(* CODESYS project CtaAppSensor_2.0.0.0.library
   Description: Sensor Library der CTA
   Version: 2.0.0.0
   Title: CtaAppSensor
   Author: SIS
   DocFormat: reStructuredText
   Placeholder: CtaAppSensor
   LanguageModelAttribute: qualified-access-only
   CompiledLibraryCompatibilityVersion: CODESYS V3.5 SP16 Patch 3
   Company: CTA
   DefaultNamespace: CtaAppSensor

Project tree, tasks and I/O mapping:
  libraries: Standard, 3.5.18.0 (System); CtaAppBmk, 2.0.0.0 (CTA); CtaAppReport, 2.0.0.0 (CTA); CtaSysConfig, 2.0.0.0 (CTA); CtaAppFilter, 1.0.0.0 (CTA); VisuSymbols, 4.5.0.0 (System); VisuDialogs, * (System); CtaSysSensorReCalculation, 1.0.0.0 (CTA); CtaVisSymbols, 2.0.0.0 (CTA); CtaAppInfluxLog, 1.0.0.1 (CTA); CtaSysIO, 2.0.0.0 (CTA); CtaVisHelp, 2.0.0.0 (CTA); CtaAppModbusSpezifikation, 1.0.0.1 (CTA); CtaVisApps, 1.0.0.0 (CTA); CtaSysFU, 2.0.0.0 (CTA)
  40 Visualizations/
    ICON/
      SENSOR_FLAT/
        SENSOR_FLAT_TXT_RIGHT/
          ABOVE/
            visualisation VIS_SENSOR_FLAT_RigthAboveCheckIsEnabled
            visualisation VIS_SENSOR_FLAT_RIGHT_ABOVE
            visualisation VIS_SENSOR_FLAT_RigthAboveCheckQuerry
          BELOW/
            visualisation VIS_SENSOR_FLAT_RIGHT_BELOW
            visualisation VIS_SENSOR_FLAT_RigthBelowCheckIsEnabled
            visualisation VIS_SENSOR_FLAT_RigthBelowCheckQuerry
          MIDDLE/
            visualisation VIS_SENSOR_FLAT_RIGHT_MIDDLE
            visualisation VIS_SENSOR_FLAT_RigthMiddleCheckIsEnabled
            visualisation VIS_SENSOR_FLAT_RigthMiddleCheckQuerry
        SENSOR_FLAT_TXT_LEFT/
          BELOW/
            visualisation VIS_SENSOR_FLAT_LEFT_BELOW
            visualisation VIS_SENSOR_FLAT_LeftBelowCheckIsEnabled
            visualisation VIS_SENSOR_FLAT_LeftBelowCheckQuerry
          ABOVE/
            visualisation VIS_SENSOR_FLAT_LeftAboveCheckQuerry
            visualisation VIS_SENSOR_FLAT_LEFT_ABOVE
            visualisation VIS_SENSOR_FLAT_LeftAboveCheckIsEnabled
          MIDDLE/
            visualisation VIS_SENSOR_FLAT_LeftMiddleCheckIsEnabled
            visualisation VIS_SENSOR_FLAT_LeftMiddleCheckQuerry
            visualisation VIS_SENSOR_FLAT_LEFT_MIDDLE
      SENSOR_BASE/
        ICON/
          Round/
            visualisation SensorRound
          Flat/
            visualisation SensorFlat
          Value/
            visualisation ValueDwnUp
            visualisation ValueUpDwn
      SENSOR_ROUND/
        SENSOR_ROUND_TXT_RIGHT/
          ABOVE/
            visualisation VIS_SENSOR_ROUND_RIGHT_ABOVE
            visualisation VIS_SENSOR_ROUND_RightAboveCheckIsEnabled
            visualisation VIS_SENSOR_ROUND_RightAboveCheckQuerry
          BELOW/
            visualisation VIS_SENSOR_ROUND_RIGHT_BELOW
            visualisation VIS_SENSOR_ROUND_RightBelowCheckQuerry
            visualisation VIS_SENSOR_ROUND_RightBelowCheckIsEnabled
        SENSOR_ROUNF_TXT_LEFT/
          ABOVE/
            visualisation VIS_SENSOR_ROUND_LEFT_ABOVE
            visualisation VIS_SENSOR_ROUND_LeftAboveCheckIsEnabled
            visualisation VIS_SENSOR_ROUND_LeftAboveCheckQuerry
          BELOW/
            visualisation VIS_SENSOR_ROUND_LEFT_BELOW
            visualisation VIS_SENSOR_ROUND_LeftBelowCheckIsEnabled
            visualisation VIS_SENSOR_ROUND_LeftBelowCheckQuerry
    POPUP/
      visualisation POPUP_SENSOR
      PARAMETER/
        visualisation VIS_SENSOR_PARAMETER
        visualisation VIS_SENSOR_PARAMETER_LISTE
        SENSOR_ParameterBase/
          visualisation VIS_SENSOR_PARAMETER_BASE0
          visualisation VIS_SENSOR_PARAMETER_BASE
        SENSOR_ReportManagement/
          visualisation Sensor_LowAlarm_Param
          visualisation Sensor_HighAlarm_Param
          visualisation Sensor_HighWarning_Param
          visualisation VIS_SENSOR_PARAMETER_REPORTMNG
          visualisation VIS_SENSOR_PARAMETER_REPORTMNG_1
          visualisation Sensor_LowWarning_Param
        SENSOR_InfluxDb/
          visualisation VIS_SENSOR_PARAMETER_TRENDLOG
          visualisation VIS_SENSOR_PARAMETER_TRENDLOG0
        SENSOR_Filter/
          visualisation VIS_SENSOR_PARAMETER_FILTER
          visualisation VIS_SENSOR_PARAMETER_FILTER_1
        IO_Parameter/
          visualisation VIS_SENSOR_IO_PARAMETER
      visualisation VIS_SENSOR_LISTE
      MANUAL/
        visualisation VIS_SENSOR_MANUAL
      OVERVIEW/
        visualisation VIS_SENSOR_OVERVIEW
        visualisation VIS_SENSOR_OVERVIEW0
      REPORTS/
        visualisation VIS_SENSOR_REPORTS
      BUS/
        visualisation Sensor_BUS_CS
        visualisation Sensor_BUS
        visualisation Sensor_BUS_SW0_Detail
        visualisation Sensor_BUS_SW1_Detail
        visualisation Sensor_BUS_SW2_Detail
        visualisation Sensor_BUS_SW3_Detail
      PLACEHOLDER/
        visualisation VIS_SENSOR_PLACEHOLDER
        visualisation VIS_SENSOR_PLACEHOLDER0
        visualisation VIS_SENSOR_PLACEHOLDER_1
        visualisation VIS_SENSOR_PLACEHOLDER0_1
  30 Program Organization Units/
    fb's/
      Sensor/
        function block fbSensor [ST]: proModulType, actReport, proITF_REPORTMANAGER, actErrorCondition, proLockDown, proAvailable, proAcknowlege, proAtIconNr, actTrendLog, proEn, proEnSymbol, metSetReal, metSetBool, proIsEnabled, proIsError, proStateSymbol, proCountedError, proCountedInfo, proCountedWarning, actState, proInvertierung, proxErrorConditionValue, proConfigError, actConfig, P_scAnalogAlarm_fbxEnableOverflowAl, P_scAnalogAlarm_fbxEnableUnderflowAl, P_scBase_fbxEnable, P_scVisu_fbusiDezimalPos, P_scAlCondition_fbxEnable, P_scAlCondition_fbtDelayTillCondition, P_scHighAlarm_fbiRetryTillLock, P_scHighAlarm_fbiTypeOfAcknolage, P_scHighAlarm_fbrHysterese, P_scHighAlarm_fbrValue, P_scHighAlarm_fbtDelayTillAlarm, P_scHighAlram_fbxDoesAlarm, P_scHighWarning_fbrValue, P_scHighWarning_fbtDelayTillWarning, P_scHighWarning_fbxDoesWarning, P_scInfluxDb_fbxEnable, P_scLoAlarm_fbiRetryTillLock, P_scLoAlarm_fbiTypeOfAcknolage, P_scLoAlarm_fbrHysterese, P_scLoAlarm_fbrValue, P_scLoAlarm_fbtDelayTillAlarm, P_scLoAlarm_fbxDoesAlarm, P_scLoWarning_fbrValue, P_scLoWarning_fbtDelayTillWarning, P_scLoWarning_fbxDoesWarning, P_scManual_fbrManualOnY, P_scManual_fbuiManualControl, P_scManual_fbuiManualState, P_scManual_fbxAllowManualOn, P_scAlarmReset_fbtDealyTillReset, P_scFilter_fbrValue, P_scFilter_fbxEnabled, proSensorITF, proRawValue, proSoftwareValue, proIsWarning, proIsHandOnOrOff, proIsReady, proHandOff, proHandOn, proHandOnY, proAuto, proManualTrue, proManualFalse, proValueInputType, metSetITF, actDigital, actAnalog, proPhysicalValue, actReCalculate, ITF_RC, actMbState, proModbusTest, proModbusStateWord, proModbusControllWord, prorValue
    fc's/
      function fcGetBigerStringValue [ST]
      AlarmControll/
        function fcHighControl [ST]
        function fcLowControl [ST]
      Visu/
        function fcCheckQuerryAndIconReturn [ST]
  00000000-0000-0000-0000-000000000000|D:\CoDeSys\LibrariesV3\trunk\Intern\CAA\CAA Template\3.4.0.0 draft\Placeholder.xml
  00000000-0000-0000-0000-000000000000|D:\CoDeSys\LibrariesV3\trunk\Intern\CAA\CAA Template\3.2.0.3 draft\Prefix.pdf
  00000000-0000-0000-0000-000000000000|D:\CoDeSys\LibrariesV3\trunk\Intern\CAA\CAA Template\3.5.2.0 draft\Placeholder.xml
  20 Structs/
    data type scParameter
    LowWarning/
      data type scLoWarning
    BASE/
      data type scBase
    Alarme/
      data type scAnalogAlarm
      Zusatzbedingungen/
        data type scAlCondition
      AlarmReset/
        data type scAlarmReset
    HighWarning/
      data type scHighWarning
    InfluxDb/
      data type scInfluxDb
    Filter/
      data type scFilter
    HighAlarm/
      data type scHighAlarm
    LowAlarm/
      data type scLoAlarm
    Manual/
      data type scManual
    data type enInputType
    Visu/
      data type scVisu
  50 Images/
  10 Documenation/
    global variables VersionHistory
    global variables readMe
  21 Interface/
    interface ITF_SENSOR: proConfigError, P_scBase_fbxEnable, P_scVisu_fbusiDezimalPos, P_scManual_fbxAllowManualOn, P_scManual_fbuiManualState, P_scManual_fbuiManualControl, P_scManual_fbrManualOnY, P_scFilter_fbxEnabled, P_scFilter_fbrValue, P_scLoWarning_fbxDoesWarning, P_scLoWarning_fbrValue, P_scLoWarning_fbtDelayTillWarning, P_scLoAlarm_fbxDoesAlarm, P_scLoAlarm_fbrValue, P_scLoAlarm_fbrHysterese, P_scLoAlarm_fbtDelayTillAlarm, P_scLoAlarm_fbiRetryTillLock, P_scLoAlarm_fbiTypeOfAcknolage, P_scHighWarning_fbxDoesWarning, P_scHighWarning_fbrValue, P_scHighWarning_fbtDelayTillWarning, P_scHighAlram_fbxDoesAlarm, P_scHighAlarm_fbrValue, P_scHighAlarm_fbrHysterese, P_scHighAlarm_fbtDelayTillAlarm, P_scHighAlarm_fbiRetryTillLock, P_scHighAlarm_fbiTypeOfAcknolage, P_scInfluxDb_fbxEnable, P_scAnalogAlarm_fbxEnableOverflowAl, P_scAnalogAlarm_fbxEnableUnderflowAl, P_scAlCondition_fbxEnable, P_scAlCondition_fbtDelayTillCondition, P_scAlarmReset_fbtDealyTillReset, proSensorITF, proCountedError, proCountedInfo, proITF_REPORTMANAGER, proCountedWarning, proRawValue, proSoftwareValue, proEnSymbol, proStateSymbol, proIsHandOnOrOff, proHandOn, proIsError, proIsWarning, proEn, proIsEnabled, proHandOff, proHandOnY, proIsReady, proAuto, proManualFalse, proManualTrue, proValueInputType, proPhysicalValue, proxErrorConditionValue, proInvertierung, prorValue, proLockDown, proAvailable, proAcknowlege, proAtIconNr, ITF_RC, proModbusStateWord, proModbusTest, proModbusControllWord
  11 Library Parameter/
  12 Konstanten/
    global variables GlobalKonstant
  60 Textlisten/
    text list GlobalTextList
    text list Info
    Types/
      text list WarnungsStatus
      text list ValueInputType
    Reports/
      text list Error
      text list Warnung
  13 Globale Variablen/
  5ce3da45-db07-42e7-a21c-a00fff4ed8f6|C:\Users\sis\Downloads\dip-switch.svg
  5ce3da45-db07-42e7-a21c-a00fff4ed8f6|C:\Users\sis\Downloads\lightning-bolt-circle.svg
  5ce3da45-db07-42e7-a21c-a00fff4ed8f6|C:\Users\sis\Downloads\sine-wave.svg
  5ce3da45-db07-42e7-a21c-a00fff4ed8f6|C:\Users\sis\Downloads\eye.svg
  5ce3da45-db07-42e7-a21c-a00fff4ed8f6|C:\Users\sis\Downloads\lan.svg
*)

// 20 Structs/scParameter
{attribute 'pack_mode' := '1'} 
TYPE scParameter :
    STRUCT
        scBase              :   scBase;
		scManual			:	scManual;
		scFilter			:	scFilter;
		scLoWarning			:	scLoWarning;
		scLoAlarm			:	scLoAlarm;
		scHighWarning		:	scHighWarning;
		scHighAlarm			:	scHighAlarm;
		scInfluxDb			:	scInfluxDb;
		scAnalogAlarm		:	scAnalogAlarm;
		scAlCondition		:	scAlCondition;
		scAlarmReset		:	scAlarmReset;
		scVisu				:	scVisu;
    END_STRUCT
END_TYPE

// 20 Structs/HighWarning/scHighWarning
TYPE scHighWarning :
	STRUCT
		fbxDoesWarning			:	CtaSysConfig.fbBOOL;
		fbrValue				:	CtaSysConfig.fbREAL;
		fbtDelayTillWarning		:	CtaSysConfig.fbTIME;	
	END_STRUCT
END_TYPE

// 20 Structs/HighAlarm/scHighAlarm
TYPE scHighAlarm :
	STRUCT
		fbxDoesAlarm			:	CtaSysConfig.fbBOOL;
		fbrValue				:	CtaSysConfig.fbREAL;
		fbrHysterese			:	CtaSysConfig.fbREAL;
		fbtDeleayTillAlarm		:	CtaSysConfig.fbTIME;
		fbiRetryTillLock		:	CtaSysConfig.fbINT;
		fbiTypeOfAcknolage		:	CtaSysConfig.fbINT;
	END_STRUCT
END_TYPE

// 20 Structs/LowAlarm/scLoAlarm
TYPE scLoAlarm :
	STRUCT
		fbxDoesAlarm			:	CtaSysConfig.fbBOOL;
		fbrValue				:	CtaSysConfig.fbREAL;
		fbrHysterese			:	CtaSysConfig.fbREAL;
		fbtDeleayTillAlarm		:	CtaSysConfig.fbTIME;
		fbiRetryTillLock		:	CtaSysConfig.fbINT;
		fbiTypeOfAcknolage		:	CtaSysConfig.fbINT;
	END_STRUCT
END_TYPE

// 20 Structs/LowWarning/scLoWarning
TYPE scLoWarning :
	STRUCT
		fbxDoesWarning			:	CtaSysConfig.fbBOOL;
		fbrValue				:	CtaSysConfig.fbREAL;
		fbtDelayTillWarning		:	CtaSysConfig.fbTIME;		
	END_STRUCT
END_TYPE

// 20 Structs/Alarme/scAnalogAlarm
TYPE scAnalogAlarm :
	STRUCT
		fbxEnableOverflowAl		:	CtaSysConfig.fbBOOL;
		fbxEnableUnderflowAl	:	CtaSysConfig.fbBOOL;
	END_STRUCT
END_TYPE

// 20 Structs/Filter/scFilter
TYPE scFilter :
	STRUCT
		fbxEnabled	:	CtaSysConfig.fbBOOL;
		fbrValue	:	CtaSysConfig.fbREAL;
	END_STRUCT
END_TYPE

// 20 Structs/BASE/scBase
{attribute 'pack_mode' := '1'} 
TYPE scBase :
    STRUCT
        fbxEnable       :   CtaSysConfig.fbBOOL;
    END_STRUCT
END_TYPE

// 20 Structs/InfluxDb/scInfluxDb
{attribute 'pack_mode' := '1'} 
TYPE scInfluxDb :
    STRUCT
        fbxEnable       :   CtaSysConfig.fbBOOL;
    END_STRUCT
END_TYPE

// 20 Structs/Alarme/Zusatzbedingungen/scAlCondition
TYPE scAlCondition :
	STRUCT
		fbxEnable				:	CtaSysConfig.fbBOOL;
		fbtDelayTillCondition	:	CtaSysConfig.fbTIME;
	END_STRUCT
END_TYPE

// 20 Structs/Alarme/AlarmReset/scAlarmReset
TYPE scAlarmReset :
	STRUCT
		fbtDelayTillReset	:	CtaSysConfig.fbTIME;		
	END_STRUCT
END_TYPE

// 20 Structs/Manual/scManual
TYPE scManual :
	STRUCT
		fbxAlowManualOn		:	CtaSysConfig.fbBOOL;
		fbuiManualState		:	CtaSysConfig.fbUINT;
		fbuiManualControl	:	CtaSysConfig.fbUINT;
		fbrManualOnY		:	CtaSysConfig.fbREAL;
	END_STRUCT
END_TYPE

// 20 Structs/enInputType
{attribute 'qualified_only'}
{attribute 'strict'}
TYPE enInputType :
(
	Default := 0,
	AnalogInput,
	DigitalInput,
	Analog_ITF_Input,
	Digital_ITF_Input	
);
END_TYPE

// 20 Structs/Visu/scVisu
TYPE scVisu :
	STRUCT
		fbusiDezimalPos		:	CtaSysConfig.fbUSINT;
	END_STRUCT
END_TYPE

// 10 Documenation/VersionHistory
(* 

.. image:: ../../Images/CTA_Logo.jpg
   :align: right
   :width: 15% 

**Vorlage**   


============ =========== =========== ============================================
**Date**     **Version** **Author**  **Change**
------------ ----------- ----------- --------------------------------------------
04.03.2021   0.0.0.0     SIS         Vorlage erstellt

============ =========== =========== ============================================


*)
VAR_GLOBAL
    stInfo : STRING:= '0.0.0.0, Vorlage, CTA';
END_VAR

// 10 Documenation/readMe
(*

**ReadMe**
 
|	**Empfehlung**
|
|	Bibliothek CtaAppSensor zur auswertung von Sensoren
|	Instanzieren Sie den CtaAppSensor.fbSensor in ihrem Funktionsbaustein oder POU beispielsweise als fbTFühlX (X = Nr.) 
|	Deklarieren Sie die Struktur Variable welche als Parameter und zur ansteuerung dienen wie im Code beispiel.
|  
| *Beispiel* 

+-----------------------+---------------------------------------------------------------------------------------------------------------------------------------------------------------------------------------------------------------------------------------------------------------------------------------------------------------------------------------------------------------------------------------------------------------------------------------+
| Beschreibung          |  Code                                                                                                                                                                                                                                                                                                                                                                                                                                 |
+=======================+=======================================================================================================================================================================================================================================================================================================================================================================================================================================+
| POU oder SmFb         | .. code-block:: codesys                                                                                                                                                                                                                                                                                                                                                                                                               |
|                       |                                                                                                                                                                                                                                                                                                                                                                                                                                       |
|                       |	// Deklaration als VAR im POU oder dem selbsterstellten Funktionsbaustein                                                                                                                                                                                                                                                                                                                                                        	|
|                       |   VAR   																																																				 																																																				|
|						|	    (*Temperaturfühler 1*)																																																		 																																																	|
|						|		fbTFühl1			: CtaAppSensor.fbSensor;                                                                                                                                                                                                                                                                                                                                                               						|
|			 			|	END_VAR                                                                                                                                                                                                                                                                                                                                                                                                                          	|
+-----------------------+---------------------------------------------------------------------------------------------------------------------------------------------------------------------------------------------------------------------------------------------------------------------------------------------------------------------------------------------------------------------------------------------------------------------------------------+
| Code für Init         | .. code-block:: codesys                                                                                                                                                                                                                                                                                                                                                                                                               |
|                       |   																																																					 																																																				|
|			 			|	// Kopieren des nachfolgenden Codes in eine Action zur Initialisierung der Parameter. Zum Beispiel actConfig.																																																				 																										|
|                       |	{region "Parameter Temperaturfühler 1"}                                                                                                                                                                                                                                                                                                                                                                                             |
|			 			|		(*Basis*)                                                                                                                                                                                                                                                                                                                                                                                                                       |
|						|		fbTFühl1.scParameter.scBase.fbxEnable                			(_WertInit :=  TRUE																		 );		//P1 Ein- Ausschalten des Sensors                                                                                                                                                                                                                               |
|						|		(*Handansteuerung*)                                                                                                                                                                                                                                                                                                                                                                                                             |
|						|		fbTFühl1.scParameter.scManual.fbxAlowManualOn					(_WertInit := FALSE																		 );     //P2 Handansteuerung zulassen / nicht zulassen                                                                                                                                                                                                                  |
|						|		fbTFühl1.scParameter.scManual.fbuiManualState					(_WertInit :=	  0									, _MinInit :=     0, _MaxInit:=     2);     //P3 Ansteuerungsmodus des Sensors (auto, manuell, gesperrt)                                                                                                                                                                                                    |
|						|		fbTFühl1.scParameter.scManual.fbuiManualControl					(_WertInit :=     0									, _MinInit :=     0, _MaxInit:=     1);     //P4 Ansteuerungsignal des Sensors (TRUE,FALSE)                                                                                                                                                                                                                 |
|						|		fbTFühl1.scParameter.scManual.fbrManualOnY						(_WertInit :=   0.0									, _MinInit :=      , _MaxInit:=      );     //P5 Manueller Stellwert für den SEnsor                                                                                                                                                                                                                         |
|						|		(*Filter*)                                                                                                                                                                                                                                                                                                                                                                                                                      |
|						|		fbTFühl1.scParameter.scFilter.fbxEnabled						(_WertInit := FALSE																		 );		//P6 Ein- Ausschalten des Filters                                                                                                                                                                                                                               |
|						|		fbTFühl1.scParameter.scFilter.fbrValue							(_WertInit :=   0.0									, _MinInit :=      , _MaxInit:=      );		//P7 Filterwert                                                                                                                                                                                                                                                 |
|						|		(*LowWarning*)                                                                                                                                                                                                                                                                                                                                                                                                                  |
|						|		fbTFühl1.scParameter.scLoWarning.fbxDoesWarning					(_WertInit := FALSE																		 );		//P8 Ein- Ausschalten der LowWarning                                                                                                                                                                                                                            |
|						|		fbTFühl1.scParameter.scLoWarning.fbrValue						(_WertInit :=   0.0									, _minInit :=      , _maxInit:= 	 );		//P9 Wert bei welcher die LowWarning ausgelöst wird                                                                                                                                                                                                             |
|						|		fbTFühl1.scParameter.scLoWarning.fbtDelayTillWarning			(_WertInit :=  T#0S									, _minInit :=      , _maxInit:=      );		//P10 Verzögerungszeit für die Ausgabe des LowWarining Fehlers                                                                                                                                                                                                  |
|						|		(*LowAlarm*)                                                                                                                                                                                                                                                                                                                                                                                                                    |
|						|		fbTFühl1.scParameter.scLoAlarm.fbxDoesAlarm						(_WertInit := FALSE																		 );		//P11 Ein- Ausschalten des LowAlarm                                                                                                                                                                                                                             |
|						|		fbTFühl1.scParameter.scLoAlarm.fbrValue							(_WertInit :=   0.0									, _minInit :=      , _maxInit:= 	 );		//P12 Wert bei welchem der LowAlarm ausgelöst wird                                                                                                                                                                                                              |
|						|		fbTFühl1.scParameter.scLoAlarm.fbrHysterese						(_WertInit :=   0.0									, _minInit :=      , _maxInit:= 	 );		//P13 Histerese welche zur Rücksetung des Fehlers erreicht werden muss                                                                                                                                                                                          |
|						|		fbTFühl1.scParameter.scLoAlarm.fbtDeleayTillAlarm				(_WertInit :=  T#0S									, _minInit :=      , _maxInit:= 	 );		//P14 Verzögerungszeit für die Ausgabe des LowAlarm Fehlers                                                                                                                                                                                                     |
|						|		fbTFühl1.scParameter.scLoAlarm.fbiTypeOfAcknolage				(_WertInit :=     0 								, _minInit :=     0, _maxInit:=     2);		//P15 Art der Quittierung des Fehlers (auto, quittierned, quittiernd bis n Meldung)                                                                                                                                                                             |
|						|		fbTFühl1.scParameter.scLoAlarm.fbiRetryTillLock					(_WertInit :=     3									, _minInit :=     0, _maxInit:=     5);		//P16 Maximale Anzahl Wiederholungen bis zu Sperrung der Anlage                                                                                                                                                                                                 |
|						|		(*HighWarning*)                                                                                                                                                                                                                                                                                                                                                                                                                 |
|						|		fbTFühl1.scParameter.scHighWarning.fbxDoesWarning				(_WertInit := FALSE																		 );		//P17 Ein- Ausschalten der HighWarning                                                                                                                                                                                                                    		|
|						|		fbTFühl1.scParameter.scHighWarning.fbrValue						(_WertInit :=   0.0									, _minInit :=      , _maxInit:= 	 );		//P18 Wert bei welcher die HighWarning ausgelöst wird                                                                                                                                                                                                     		|
|						|		fbTFühl1.scParameter.scHighWarning.fbtDelayTillWarning			(_WertInit :=  T#0S									, _minInit := 	   , _maxInit:= 	 );		//P19 Verzögerungszeit für die Ausgabe des HighWarining Fehlers                                                                                                                                                                                           		|
|						|		(*HighAlarm*)                                                                                                                                                                                                                                                                                                                                                                                                                   |
|						|		fbTFühl1.scParameter.scHighAlarm.fbxDoesAlarm					(_WertInit := FALSE															 			 );		//P20 Ein- Ausschalten des HighAlarm                                                                                                                                                                                                                            |
|						|		fbTFühl1.scParameter.scHighAlarm.fbrValue						(_WertInit :=   0.0									, _minInit :=      , _maxInit:=      );		//P21 Wert bei welchem der HighAlarm ausgelöst wird                                                                                                                                                                                                             |
|						|		fbTFühl1.scParameter.scHighAlarm.fbrHysterese					(_WertInit :=   0.0									, _minInit :=      , _maxInit:= 	 );		//P22 Histerese welche zur Rücksetung des Fehlers erreicht werden muss                                                                                                                                                                                          |
|						|		fbTFühl1.scParameter.scHighAlarm.fbtDeleayTillAlarm				(_WertInit :=  T#0S									, _minInit :=      , _maxInit:=      );		//P23 Verzögerungszeit für die Ausgabe des HighAlarm Fehlers                                                                                                                                                                                                    |
|						|		fbTFühl1.scParameter.scHighAlarm.fbiTypeOfAcknolage				(_WertInit := 	  0 								, _minInit :=      , _maxInit:=     2);		//P24 Art der Quittierung des Fehlers (auto, quittierned, quittiernd bis n Meldung)                                                                                                                                                                             |
|						|		fbTFühl1.scParameter.scHighAlarm.fbiRetryTillLock				(_WertInit :=     3									, _minInit :=      , _maxInit:=     5);		//P25 Maximale Anzahl Wiederholungen bis zu Sperrung der Anlage                                                                                                                                                                                                 |
|						|		(*Überlauf, Unterlauf*)                                                                                                                                                                                                                                                                                                                                                                                                         |
|						|		fbTFühl1.scParameter.scAnalogAlarm.fbxEnableOverflowAl			(_WertInit :=  TRUE																		 );		//P26 Ein- Ausschalten des Überlauf- Alarms                                                                                                                                                                                                                     |
|						|		fbTFühl1.scParameter.scAnalogAlarm.fbxEnableUnderflowAl			(_WertInit :=  TRUE																		 );		//P27 Ein- Ausschalten des Unterlauf- Alrams                                                                                                                                                                                                                    |
|						|		(*Zusatzbedingung*)                                                                                                                                                                                                                                                                                                                                                                                                             |
|						|		fbTFühl1.scParameter.scAlCondition.fbxEnable 					(_WertInit := FALSE																		 );		//P28 Ein- Ausschalten der Zusatzbedingung                                                                                                                                                                                                                      |
|						|		fbTFühl1.scParameter.scAlCondition.fbtDelayTillCondition		(_WertInit :=  T#0S									, _minInit :=      ,_maxInit:=       );		//P29 Verzögerung für die Zusatzbedingung                                                                                                                                                                                                                       |
|						|		(*Alarmrücksetzung*)                                                                                                                                                                                                                                                                                                                                                                                                            |
|						|		fbTFühl1.scParameter.scAlarmReset.fbtDelayTillReset				(_WertInit := T#24H									, _minInit :=      ,_maxInit:=       );		//P30 Verzögerung für die Fehlerrücksetzung                                                                                                                                                                                                                     |
|						|		(*Trendlog*)                                                                                                                                                                                                                                                                                                                                                                                                                    |
|						|		fbTFühl1.scParameter.scInfluxDb.fbxEnable            			(_WertInit := TRUE																		 );		//P31 Aktiverung / Deaktivierung der Trenddaten														 																																							|
|						|		(*Visu*)                                                                                                                                                                                                                                                                                                                                                                                                                    	|
|						|		fbTFühl1.scParameter.scVisu.fbusiDezimalPos            			(_WertInit :=     1									, _minInit := 0     , _maxInit:=    3);		//P32 Dezimalstellen auf Visu													 																																												|
|						|	{endregion}                                                                                                                                                      																																																																    | 
|						|																																																																																																										|
+-----------------------+---------------------------------------------------------------------------------------------------------------------------------------------------------------------------------------------------------------------------------------------------------------------------------------------------------------------------------------------------------------------------------------------------------------------------------------+
*)                                                                                                                                                                                                                                                                                                                                                                                                                                                               
VAR_GLOBAL
	xReadMeDone              :   BOOL; 
END_VAR

// 12 Konstanten/GlobalKonstant
{attribute 'qualified_only'}
VAR_GLOBAL CONSTANT 	
	stReportTextListError   : CtaAppReport.stReportTextList := 'CtaAppSensor.Error';
	stReportTextListWarning : CtaAppReport.stReportTextList := 'CtaAppSensor.Warnung';
	stReportTextListInfo    : CtaAppReport.stReportTextList := 'CtaAppSensor.Info';	
END_VAR

// 30 Program Organization Units/fb's/Sensor/fbSensor
FUNCTION_BLOCK fbSensor EXTENDS CtaAppBmk.fbBMK IMPLEMENTS ITF_SENSOR 
VAR_INPUT
    xAlCondition               	:   BOOL;
	xEnHandMode					:	BOOL;
 	rSimValue					:	REAL;
END_VAR                         
VAR_OUTPUT 
    xValue                      :   BOOL;
    rValue						:   REAL;
	rValueRC					:	REAL;
	xIsHandMode					:	BOOL;
END_VAR                 
VAR 
	(*Inputs*)
	ITF_IO_IN					:	CtaSysIO.ITF_IO;
	xValueIn					:	BOOL;
	rValueIn					:	REAL;	
	(* Input Type*)
	xIsITF						:	BOOL;
	xIsBool						:	BOOL;
	xIsReal						:	BOOL;
    stAlternateUnit				:	STRING(5);                
    (* State Intern*)
	xIsDigital					:	BOOL;
	_ITF_DI						: 	CtaSysIO.ITF_DI;
	_ITF_AI						:	CtaSysIO.ITF_AI; 	
	rValueTemp					:	REAL;
	xValueTemp					:	BOOL;
	enValueInputType			:   enInputType;     
    scEWI                       :   CtaAppReport.scReportNr; 
	xIsEnabled					:	BOOL;                
	xConfigError                :   BOOL;
	uiIconNr					:	UINT;
	xOk							:	BOOL;
	(* Modbus *)
    xModbusTest                 :   BOOL;
    ayMbControllWord            :   ARRAY[0..3] OF WORD;
    ayMbStateWord               :   ARRAY[0..3] OF WORD;	
    (* Parameter *)
    fbConfigFile                :   CtaSysConfig.fbConfigFile;
    scParameter                 :   scParameter;	
    (* Reports *)		
    fbReportManager			    :   CtaAppReport.fbReportManager;      
    difor					    :	DINT;                                                                    
    ayErrorReporter				:	ARRAY[1..7] OF CtaAppReport.fbReporter;
	ayWarningReporter			:	ARRAY[1..6] OF CtaAppReport.fbReporter; 	
	_xIsWarning					:	BOOL;
	xIsWarning					:	BOOL;	
	_xIsError					:	BOOL;
	xIsError					:	BOOL;		
	xLoWarning					:	BOOL;
	xLoAlarm					:	BOOL;
	xHiWarning					:	BOOL;
	xHiAlarm					:	BOOL;	
	(* Trendlogs *)
	fbTrendxValue				:	CtaAppInfluxLog.FB_LOG_NODE_BOOL;
	fbTrendrValue				:	CtaAppInfluxLog.FB_LOG_NODE_REAL;
	fbTrendrVaueUnfiltered		:	CtaAppInfluxLog.FB_LOG_NODE_REAL;
	fbTrendrVaueRC				:	CtaAppInfluxLog.FB_LOG_NODE_REAL;
	(* Filter *)
	fbFilter					:	CtaAppFilter.fbImpulsFilter;	
	rValueUngefiltert			:	REAL;	
    (* Collector *)
    diArrayPosition             :   DINT;
	xManualValue				:	BOOL;
	xIsHandOff					:	BOOL;
	xIsHandOn					:	BOOL;
	xIsAuto						:	BOOL;
	xIsHand						:	BOOL;
	TON_DelayAlCondition		: 	TON;
	xErrorConditionOn			: 	BOOL;
	(*Calculator *)				
	ITF_RC_QUERY				:	CtaSysSensorReCalculation.ITF_SENSOR_RE_CALCULATE;
END_VAR

(* Config *)
actConfig();

(* Sensor Command *)
IF xIsEnabled AND NOT xConfigError THEN
	IF xIsITF THEN
		IF __QUERYINTERFACE(ITF_IO_IN,_ITF_DI) THEN
			enValueInputType := enInputType.Digital_ITF_Input;
			actDigital();
		ELSIF __QUERYINTERFACE(ITF_IO_IN,_ITF_AI) THEN
			enValueInputType := enInputType.Analog_ITF_Input;
			actAnalog();
		END_IF
		
	ELSIF xIsBool THEN
		enValueInputType := enInputType.DigitalInput;
		actDigital();
	ELSIF xIsReal THEN
		enValueInputType := enInputType.AnalogInput;
		actAnalog();
	ELSE
		enValueInputType := enInputType.Default;		
	END_IF	
	
	(* Al Condition *)
    actErrorCondition();	
    (* EWI *)
    actReport();    

	(* Recalculation *)
	actReCalculate();             
ELSE
    IF xConfigError THEN
        (* EWI *)
      actReport();         
	END_IF;
END_IF;

(* State *)
actState();
actMbState();
(* InfluxDB *)
actTrendLog();

PROPERTY proModulType : CtaSysIO.enIOType
GET
proModulType := ITF_IO_IN.IO_TYPE;
END_GET
END_PROPERTY

ACTION actReport:
(* EWI Manager *)
fbReportManager(	stErrorInitReportTextListIn		:=	ADR(GlobalKonstant.stReportTextListError),
					stWarningInitReportTextListIn	:=	ADR(GlobalKonstant.stReportTextListWarning),
					stInfoInitReportTextListIn		:=	ADR(GlobalKonstant.stReportTextListInfo),
					scReportNr						:=	scEWI);

IF xIsBool OR (xIsITF AND __QUERYINTERFACE (ITF_IO_IN,_ITF_DI))  THEN
	(* Errors *)                        
        (* Alarm Minimalwert erreicht *)
        ayErrorReporter[1].proPrio  := 2;
        ayErrorReporter[1].metReport(     		xSetReportIn					:= xErrorConditionOn AND scParameter.scLoAlarm.fbxDoesAlarm.proValue AND xLoAlarm,
												iReportID						:= 1,
												enReportTypeIn					:= CtaAppReport.enReportType.Error,  
												enReportAcknowledgeTypeIn   	:= scParameter.scLoAlarm.fbiTypeOfAcknolage.proValue,
												tDelay							:= scParameter.scLoAlarm.fbtDeleayTillAlarm.proValue, 
												ITF_BMK_IN						:= THIS^,			              
												pstReportTextListIn				:= ADR(GlobalKonstant.stReportTextListError),
												stOptionalReportText		    := '',   
												iRetryTilReportLock 		    := scParameter.scLoAlarm.fbiRetryTillLock.proValue, 
												xResetCount         		    := FALSE,  
												tReset						    := scParameter.scAlarmReset.fbtDelayTillReset.proValue); 		

        (* Alarm Maximalwert erreicht *)    
        ayErrorReporter[2].proPrio  := 2;
        ayErrorReporter[2].metReport(     		xSetReportIn					:= xErrorConditionOn AND scParameter.scHighAlarm.fbxDoesAlarm.proValue AND xHiAlarm,
												iReportID						:= 2,
												enReportTypeIn					:= CtaAppReport.enReportType.Error,  
												enReportAcknowledgeTypeIn   	:= scParameter.scHighAlarm.fbiTypeOfAcknolage.proValue,
												tDelay							:= scParameter.scHighAlarm.fbtDeleayTillAlarm.proValue, 
												ITF_BMK_IN						:= THIS^,			              
												pstReportTextListIn				:= ADR(GlobalKonstant.stReportTextListError),
												stOptionalReportText		    := '',   
												iRetryTilReportLock 		    := scParameter.scHighAlarm.fbiRetryTillLock.proValue,
												xResetCount         		    := FALSE, 
	                               				tReset						    := scParameter.scAlarmReset.fbtDelayTillReset.proValue); 		

(* Warnungen *)      
        (* Warnung Minimalwert erreicht *)      
        ayWarningReporter[1].proPrio := 2;
        ayWarningReporter[1].metReport(			xSetReportIn					:= xErrorConditionOn AND scParameter.scLoWarning.fbxDoesWarning.proValue AND xLoWarning,
												iReportID						:= 1,
												enReportTypeIn					:= CtaAppReport.enReportType.Warning,  
												enReportAcknowledgeTypeIn   	:= CtaAppReport.enReportAcknowledgeType.Auto,
												tDelay							:= scParameter.scLoWarning.fbtDelayTillWarning.proValue, 
												ITF_BMK_IN						:= THIS^,			              
												pstReportTextListIn				:= ADR(GlobalKonstant.stReportTextListWarning),
												stOptionalReportText		    := '',   
												iRetryTilReportLock 		    := 0, 
												xResetCount         		    := FALSE,  
												tReset						    := T#0S);                       
                                  
        (* Warnung Maxiwalwert erreicht *)
        ayWarningReporter[2].proPrio := 2;
        ayWarningReporter[2].metReport(			xSetReportIn					:= xErrorConditionOn AND scParameter.scHighWarning.fbxDoesWarning.proValue AND xHiWarning,
												iReportID						:= 2,
												enReportTypeIn					:= CtaAppReport.enReportType.Warning,  
												enReportAcknowledgeTypeIn   	:= CtaAppReport.enReportAcknowledgeType.Auto,
												tDelay							:= scParameter.scHighWarning.fbtDelayTillWarning.proValue, 
												ITF_BMK_IN						:= THIS^,			              
												pstReportTextListIn				:= ADR(GlobalKonstant.stReportTextListWarning),
												stOptionalReportText		    := '',   
												iRetryTilReportLock 		    := 0, 
												xResetCount         		    := FALSE,
												tReset						    := T#0S);  
		
ELSIF xIsReal OR (xIsITF AND __QUERYINTERFACE (ITF_IO_IN,_ITF_AI)) THEN
(* Errors *)                        
	(* Alarm Minimalwert erreicht *)
	ayErrorReporter[3].proPrio  := 2;
	ayErrorReporter[3].metReport(     		xSetReportIn					:= xErrorConditionOn AND scParameter.scLoAlarm.fbxDoesAlarm.proValue AND xLoAlarm,
											iReportID						:= 3,
											enReportTypeIn					:= CtaAppReport.enReportType.Error,  
											enReportAcknowledgeTypeIn   	:= scParameter.scLoAlarm.fbiTypeOfAcknolage.proValue,
											tDelay							:= scParameter.scLoAlarm.fbtDeleayTillAlarm.proValue, 
											ITF_BMK_IN						:= THIS^,			              
											pstReportTextListIn				:= ADR(GlobalKonstant.stReportTextListError),
											stOptionalReportText		    := '',   
											iRetryTilReportLock 		    := scParameter.scLoAlarm.fbiRetryTillLock.proValue, 
											xResetCount         		    := FALSE,  
											tReset						    := scParameter.scAlarmReset.fbtDelayTillReset.proValue); 		

	(* Alarm Maximalwert erreicht *)    
	ayErrorReporter[4].proPrio  := 2;
	ayErrorReporter[4].metReport(     		xSetReportIn					:= xErrorConditionOn AND scParameter.scHighAlarm.fbxDoesAlarm.proValue AND xHiAlarm,
											iReportID						:= 4,
											enReportTypeIn					:= CtaAppReport.enReportType.Error,  
											enReportAcknowledgeTypeIn   	:= scParameter.scHighAlarm.fbiTypeOfAcknolage.proValue,
											tDelay							:= scParameter.scHighAlarm.fbtDeleayTillAlarm.proValue, 
											ITF_BMK_IN						:= THIS^,			              
											pstReportTextListIn				:= ADR(GlobalKonstant.stReportTextListError),
											stOptionalReportText		    := '',   
											iRetryTilReportLock 		    := scParameter.scHighAlarm.fbiRetryTillLock.proValue,
											xResetCount         		    := FALSE, 
											tReset						    := scParameter.scAlarmReset.fbtDelayTillReset.proValue); 
		
		(* Additional errors over interface*)
		IF NOT xIsReal THEN									
			(* Alarm Unterlauf *)
			ayErrorReporter[5].proPrio  := 2;
			ayErrorReporter[5].metReport(     		xSetReportIn					:= scParameter.scAnalogAlarm.fbxEnableUnderflowAl.proValue AND _ITF_AI.proAlUnterlauf,
													iReportID						:= 5,
													enReportTypeIn					:= CtaAppReport.enReportType.Error,  
													enReportAcknowledgeTypeIn   	:= CtaAppReport.enReportAcknowledgeType.Auto,
													tDelay							:= T#0S, 
													ITF_BMK_IN						:= THIS^,			              
													pstReportTextListIn				:= ADR(GlobalKonstant.stReportTextListError),
													stOptionalReportText		    := '',   
													iRetryTilReportLock 		    := 0, 
													xResetCount         		    := FALSE,  
													tReset						    := T#0S); 		
		
			(* Alarm Überlauf *)    
			ayErrorReporter[6].proPrio  := 2;
			ayErrorReporter[6].metReport(     		xSetReportIn					:= scParameter.scAnalogAlarm.fbxEnableOverflowAl.proValue AND _ITF_AI.proAlUeberlauf,
													iReportID						:= 6,
													enReportTypeIn					:= CtaAppReport.enReportType.Error,  
													enReportAcknowledgeTypeIn   	:= CtaAppReport.enReportAcknowledgeType.Auto,
													tDelay							:= T#0S, 
													ITF_BMK_IN						:= THIS^,			              
													pstReportTextListIn				:= ADR(GlobalKonstant.stReportTextListError),
													stOptionalReportText		    := '',   
													iRetryTilReportLock 		    := 0,
													xResetCount         		    := FALSE, 
													tReset						    := T#0S);
		END_IF
			
(* Warnungen *)      
	(* Warnung Minimalwert erreicht *)      
	ayWarningReporter[3].proPrio := 2;
	ayWarningReporter[3].metReport(			xSetReportIn					:= xErrorConditionOn AND scParameter.scLoWarning.fbxDoesWarning.proValue AND xLoWarning,
											iReportID						:= 3,
											enReportTypeIn					:= CtaAppReport.enReportType.Warning,  
											enReportAcknowledgeTypeIn   	:= CtaAppReport.enReportAcknowledgeType.Auto,
											tDelay							:= scParameter.scLoWarning.fbtDelayTillWarning.proValue, 
											ITF_BMK_IN						:= THIS^,			              
											pstReportTextListIn				:= ADR(GlobalKonstant.stReportTextListWarning),
											stOptionalReportText		    := '',   
											iRetryTilReportLock 		    := 0, 
											xResetCount         		    := FALSE,  
											tReset						    := T#0S);                       
							  
	(* Warnung Maxiwalwert erreicht *)
	ayWarningReporter[4].proPrio := 2;
	ayWarningReporter[4].metReport(			xSetReportIn					:= xErrorConditionOn AND scParameter.scHighWarning.fbxDoesWarning.proValue AND xHiWarning,
											iReportID						:= 4,
											enReportTypeIn					:= CtaAppReport.enReportType.Warning,  
											enReportAcknowledgeTypeIn   	:= CtaAppReport.enReportAcknowledgeType.Auto,
											tDelay							:= scParameter.scHighWarning.fbtDelayTillWarning.proValue, 
											ITF_BMK_IN						:= THIS^,			              
											pstReportTextListIn				:= ADR(GlobalKonstant.stReportTextListWarning),
											stOptionalReportText		    := '',   
											iRetryTilReportLock 		    := 0, 
											xResetCount         		    := FALSE,
											tReset						    := T#0S);
END_IF

(* Config Error *)    
ayErrorReporter[7].proPrio  := 1;
ayErrorReporter[7].metReport(     		xSetReportIn					:= xConfigError,
										iReportID						:= 7,
										enReportTypeIn					:= CtaAppReport.enReportType.Error,  
										enReportAcknowledgeTypeIn   	:= CtaAppReport.enReportacknowledgeType.Quit,
										tDelay							:= T#1S, 
										ITF_BMK_IN						:= THIS^,			              
										pstReportTextListIn				:= ADR(GlobalKonstant.stReportTextListError),
										stOptionalReportText		    := '',   
										iRetryTilReportLock 		    := 0, 
										xResetCount         		    := FALSE,  
										tReset						    := T#24H);                            

		
(* Warnung Hand Aus *)      
ayWarningReporter[5].proPrio := 3;  
ayWarningReporter[5].proHandLokal :=    xIsHandOff; 
ayWarningReporter[5].metReport(			xSetReportIn					:= xIsHandOff,
										iReportID						:= 5,
										enReportTypeIn					:= CtaAppReport.enReportType.Warning,  
										enReportAcknowledgeTypeIn   	:= CtaAppReport.enReportAcknowledgeType.Auto,
										tDelay							:= T#0S, 
										ITF_BMK_IN						:= THIS^,			              
										pstReportTextListIn				:= ADR(GlobalKonstant.stReportTextListWarning),
										stOptionalReportText		    := '',   
										iRetryTilReportLock 		    := 0, 
										xResetCount         		    := FALSE,  
										tReset						    := T#24H);                                  
                                
(* Warnung Hand Ein *)    
ayWarningReporter[6].proPrio := 3; 
ayWarningReporter[6].proHandLokal :=    xIsHandOn;
ayWarningReporter[6].metReport(			xSetReportIn					:= xIsHandOn OR xIsHandMode,
										iReportID						:= 6,
										enReportTypeIn					:= CtaAppReport.enReportType.Warning,  
										enReportAcknowledgeTypeIn   	:= CtaAppReport.enReportAcknowledgeType.Auto,
										tDelay							:= T#0S, 
										ITF_BMK_IN						:= THIS^,			              
										pstReportTextListIn				:= ADR(GlobalKonstant.stReportTextListWarning),
										stOptionalReportText		    := '',   
										iRetryTilReportLock 		    := 0, 
										xResetCount         		    := FALSE,  
										tReset						    := T#24H);                                           
	
(* Sync Reports *)                                         
FOR difor := LOWER_BOUND(ayErrorReporter,1) TO UPPER_BOUND(ayErrorReporter,1) DO
	fbReportManager.metSyncReporter(ayErrorReporter[difor]);	
END_FOR;
FOR difor := LOWER_BOUND(ayWarningReporter,1) TO UPPER_BOUND(ayWarningReporter,1) DO
	fbReportManager.metSyncReporter(ayWarningReporter[difor]);	
END_FOR;
                                                                          
_xIsError   := scEWI.iError <> 0;
_xIsWarning := scEWI.iWarning <> 0;
END_ACTION

PROPERTY proITF_REPORTMANAGER : CtaAppReport.ITF_REPORTMANAGER
GET
proITF_REPORTMANAGER := fbReportManager;
END_GET
END_PROPERTY

ACTION actErrorCondition:
//  Zeitverzögerung bis die Alarmierung Freigegeben wird


IF scParameter.scAlCondition.fbxEnable.proValue			THEN
	TON_DelayAlCondition(   PT:=    scParameter.scAlCondition.fbtDelayTillCondition.proValue,
							IN:=	xAlCondition,
							Q=>     xErrorConditionOn);  
             
ELSE
xErrorConditionOn		:=TRUE;	
END_IF
END_ACTION

{attribute 'monitoring' := 'variable'}
PROPERTY proLockDown : BOOL
GET
proLockDown := proIsError;
END_GET
END_PROPERTY

{attribute 'monitoring' := 'variable'}
PROPERTY proAvailable : BOOL
GET
proAvailable := proIsReady;
END_GET
END_PROPERTY

{attribute 'monitoring' := 'variable'}
PROPERTY proAcknowlege : BOOL
GET
proAcknowlege := xValue AND NOT proIsError ;
END_GET
END_PROPERTY

PROPERTY proAtIconNr : UINT
SET
uiIconNr := proAtIconNr;
END_SET
GET
proAtIconNr:= uiIconNr;
END_GET
END_PROPERTY

ACTION actTrendLog:
(* Istwert bool *)
fbTrendxValue.ENABLE		:= 	scParameter.scBase.fbxEnable.proValue AND 
								scParameter.scInfluxDb.fbxEnable.proValue;
fbTrendxValue.KEY           :=  CONCAT(stObjID,'_xValue');
fbTrendxValue.SET_VALUE     :=  xValue;

(* Istwert real *)
fbTrendrValue.ENABLE		:=	scParameter.scBase.fbxEnable.proValue AND 
								scParameter.scInfluxDb.fbxEnable.proValue;
fbTrendrValue.KEY           :=  CONCAT(stObjID,'_rValue');
fbTrendrValue.SET_VALUE     :=  rValue;

IF (xIsITF AND  __QUERYINTERFACE (ITF_IO_IN,_ITF_AI)) OR xIsReal THEN
	(* Istwert real ungefiltert*)
	fbTrendrVaueUnfiltered.ENABLE		:=	scParameter.scBase.fbxEnable.proValue AND 
											scParameter.scInfluxDb.fbxEnable.proValue;
	fbTrendrVaueUnfiltered.KEY			:=  CONCAT(stObjID,'_rValueUnfiltered');
	fbTrendrVaueUnfiltered.SET_VALUE	:= 	rValueUngefiltert;
ELSE
	(* Istwert real ungefiltert*)
	fbTrendrVaueUnfiltered.ENABLE		:=	FALSE;
	fbTrendrVaueUnfiltered.KEY			:=  CONCAT(stObjID,'_rValueUnfiltered');
	fbTrendrVaueUnfiltered.SET_VALUE	:= 	rValueUngefiltert;	
END_IF;

IF __QUERYINTERFACE(ITF_RC_QUERY,ITF_RC_QUERY) THEN
	(* Recalculatet Value Enable*)
	fbTrendrVaueRC.ENABLE				:=	scParameter.scBase.fbxEnable.proValue AND 
											scParameter.scInfluxDb.fbxEnable.proValue;
	fbTrendrVaueRC.KEY					:=  CONCAT(stObjID,'_rValueRecalculatet');
	fbTrendrVaueRC.SET_VALUE			:= 	rValueRC;
ELSE
	(* Recalculatet Value Disable*)
	fbTrendrVaueRC.ENABLE				:=	FALSE;
	fbTrendrVaueRC.KEY					:=  CONCAT(stObjID,'_rValueRecalculatet');
	fbTrendrVaueRC.SET_VALUE			:= 	rValueRC;	
END_IF;
END_ACTION

PROPERTY proEn : BOOL
SET
xIsEnabled := proEn;
END_SET
GET
proEn := xIsEnabled;
END_GET
END_PROPERTY

PROPERTY proEnSymbol : STRING
GET
IF xIsEnabled THEN
    proEnSymbol := 'CtaVisSymbols.ImagePool.CheckboxChecked_blue';
ELSE    
    proEnSymbol := 'CtaVisSymbols.ImagePool.CheckboxUnchecked_withe'; 
END_IF;
END_GET
END_PROPERTY

METHOD metSetReal
VAR_INPUT
	rRealIn				:	REAL;
	stAlternateUnitIn	:	STRING(5);
END_VAR
rValueIn 		:= rRealIn;
xIsITF 			:= FALSE;
xIsBool 		:= FALSE;
xIsReal 		:= TRUE;
stAlternateUnit := stAlternateUnitIn;
END_METHOD

METHOD metSetBool
VAR_INPUT
	xBoolIn		:  BOOL;
END_VAR
xValueIn := xBoolIn;
xIsITF	:= FALSE;
xIsBool := TRUE;
xIsReal := FALSE;
END_METHOD

PROPERTY proIsEnabled : BOOL
GET
proIsEnabled := xIsEnabled;
END_GET
END_PROPERTY

PROPERTY proIsError : BOOL
GET
proIsError := xIsError;
END_GET
END_PROPERTY

PROPERTY proStateSymbol : STRING
GET
IF xIsError THEN
    proStateSymbol := 'CtaVisSymbols.ImagePool.CtaError';
ELSE    
    IF xIsWarning THEN
        IF scEWI.iWarning = 5 THEN
            proStateSymbol := 'CtaVisSymbols.ImagePool.front_hand_Yellow_Off';
        ELSIF scEWI.iWarning = 6 THEN
            proStateSymbol := 'CtaVisSymbols.ImagePool.front_hand_Yellow';
        ELSE
            proStateSymbol := 'CtaVisSymbols.ImagePool.CtaWarning';
        END_IF;
     ELSE
         proStateSymbol := '';
	 END_IF
END_IF;
END_GET
END_PROPERTY

PROPERTY proCountedError : INT
GET
proCountedError := fbReportManager.proAnzError;
END_GET
END_PROPERTY

PROPERTY proCountedInfo : INT
GET
proCountedInfo := fbReportManager.proAnzInfo;
END_GET
END_PROPERTY

PROPERTY proCountedWarning : INT
GET
proCountedWarning := fbReportManager.proAnzWarning;
END_GET
END_PROPERTY

ACTION actState:
xIsWarning      := _xIsWarning;         
xIsError        := _xIsError;        
xIsEnabled      := scParameter.scBase.fbxEnable.proValue;         
xIsHandOn       := scParameter.scManual.fbuiManualState.proValue = 2;         
xIsHandOff      := scParameter.scManual.fbuiManualState.proValue = 1;          
xIsAuto         := scParameter.scManual.fbuiManualState.proValue = 0;
xManualValue	:= scParameter.scManual.fbuiManualControl.proValue = 1 AND scParameter.scManual.fbuiManualControl.proValue <> 0;
xIsHand        	:= xIsHandOn OR xEnHandMode OR xIsHandOff;
END_ACTION

PROPERTY proInvertierung : BOOL;
GET
IF __QUERYINTERFACE(_ITF_DI,_ITF_DI) THEN	
	proInvertierung := 	TO_BOOL(CtaSysConfig.fcGetEnumerationId(_ITF_DI.P_scfbDI_fbxInvert));
ELSE
	proInvertierung := FALSE;
END_IF
END_GET
END_PROPERTY

PROPERTY proxErrorConditionValue : BOOL
GET
proxErrorConditionValue := xErrorConditionOn;
END_GET
END_PROPERTY

PROPERTY proConfigError : BOOL
GET
proConfigError := xConfigError;
END_GET
END_PROPERTY

ACTION actConfig:
(* Config Fb *)
fbConfigFile();

(* Base Parameter *)
scParameter.scBase.fbxEnable                			(_usiParaNr :=  1, ItfConfigFb := fbConfigFile);

(* Manual *)
scParameter.scManual.fbxAlowManualOn					(_usiParaNr :=  2, itfConfigFb := fbConfigFile);
scParameter.scManual.fbuiManualState					(_usiParaNr :=  3, itfConfigFb := fbConfigFile);
scParameter.scManual.fbuiManualControl					(_usiParaNr :=  4, itfConfigFb := fbConfigFile);
scParameter.scManual.fbrManualOnY						(_usiParaNr :=  5, itfConfigFb := fbConfigFile);

(* Filter *)
scParameter.scFilter.fbxEnabled							(_usiParaNr :=  6, itfConfigFb := fbConfigFile);
scParameter.scFilter.fbrValue							(_usiParaNr :=  7, itfConfigFb := fbConfigFile);

(* Low warning *)
scParameter.scLoWarning.fbxDoesWarning					(_usiParaNr :=  8, itfConfigFb := fbConfigFile);
scParameter.scLoWarning.fbrValue						(_usiParaNr :=  9, itfConfigFb := fbConfigFile);
scParameter.scLoWarning.fbtDelayTillWarning				(_usiParaNr := 10, itfConfigFb := fbConfigFile);

(* Low alarm *)
scParameter.scLoAlarm.fbxDoesAlarm						(_usiParaNr := 11, itfConfigFb := fbConfigFile);
scParameter.scLoAlarm.fbrValue							(_usiParaNr := 12, itfConfigFb := fbConfigFile);
scParameter.scLoAlarm.fbrHysterese						(_usiParaNr := 13, itfConfigFb := fbConfigFile);
scParameter.scLoAlarm.fbtDeleayTillAlarm				(_usiParaNr := 14, itfConfigFb := fbConfigFile);
scParameter.scLoAlarm.fbiTypeOfAcknolage				(_usiParaNr := 15, itfConfigFb := fbConfigFile, _MinInit := 0 , _MaxInit := 2);
scParameter.scLoAlarm.fbiRetryTillLock					(_usiParaNr := 16, itfConfigFb := fbConfigFile);

(* High warning *)
scParameter.scHighWarning.fbxDoesWarning				(_usiParaNr := 17, itfConfigFb := fbConfigFile);
scParameter.scHighWarning.fbrValue						(_usiParaNr := 18, itfConfigFb := fbConfigFile);
scParameter.scHighWarning.fbtDelayTillWarning			(_usiParaNr := 19, itfConfigFb := fbConfigFile);

(* High alarm *)
scParameter.scHighAlarm.fbxDoesAlarm					(_usiParaNr := 20, itfConfigFb := fbConfigFile);
scParameter.scHighAlarm.fbrValue						(_usiParaNr := 21, itfConfigFb := fbConfigFile);
scParameter.scHighAlarm.fbrHysterese					(_usiParaNr := 22, itfConfigFb := fbConfigFile);
scParameter.scHighAlarm.fbtDeleayTillAlarm				(_usiParaNr := 23, itfConfigFb := fbConfigFile);
scParameter.scHighAlarm.fbiTypeOfAcknolage				(_usiParaNr := 24, itfConfigFb := fbConfigFile, _MinInit := 0 , _MaxInit := 2);
scParameter.scHighAlarm.fbiRetryTillLock				(_usiParaNr := 25, itfConfigFb := fbConfigFile);

(* Alarm *)
scParameter.scAnalogAlarm.fbxEnableOverflowAl			(_usiParaNr := 26, itfConfigFb := fbConfigFile);
scParameter.scAnalogAlarm.fbxEnableUnderflowAl			(_usiParaNr := 27, itfConfigFb := fbConfigFile);

(* Alarm extra conditions *)
scParameter.scAlCondition.fbxEnable 					(_usiParaNr := 28, itfConfigFb := fbConfigFile);
scParameter.scAlCondition.fbtDelayTillCondition			(_usiParaNr := 29, itfConfigFb := fbConfigFile);

(* Alarm reset after... *)
scParameter.scAlarmReset.fbtDelayTillReset				(_usiParaNr := 30, itfConfigFb := fbConfigFile);

(* InfluxDb *)
scParameter.scInfluxDb.fbxEnable            			(_usiParaNr := 31, ItfConfigFb := fbconfigFile);

(* Visu *)
scParameter.scVisu.fbusiDezimalPos						(_usiParaNr := 32, ItfConfigFb := fbconfigFile, _minInit := 0, _maxInit := 3);

xConfigError := fbConfigFile.xError;
END_ACTION

PROPERTY P_scAnalogAlarm_fbxEnableOverflowAl : CtaSysConfig.ITF_DATATYPE
GET
P_scAnalogAlarm_fbxEnableOverflowAl:= scParameter.scAnalogAlarm.fbxEnableOverflowAl;
END_GET
END_PROPERTY

PROPERTY P_scAnalogAlarm_fbxEnableUnderflowAl : CtaSysConfig.ITF_DATATYPE
GET
P_scAnalogAlarm_fbxEnableUnderflowAl := scParameter.scAnalogAlarm.fbxEnableUnderflowAl;
END_GET
END_PROPERTY

PROPERTY P_scBase_fbxEnable : CtaSysConfig.ITF_DATATYPE
GET
P_scBase_fbxEnable := scParameter.scBase.fbxEnable;
END_GET
END_PROPERTY

PROPERTY P_scVisu_fbusiDezimalPos : CtaSysConfig.ITF_DATATYPE
GET
P_scVisu_fbusiDezimalPos := scParameter.scVisu.fbusiDezimalPos;
END_GET
END_PROPERTY

PROPERTY P_scAlCondition_fbxEnable : CtaSysConfig.ITF_DATATYPE
GET
P_scAlCondition_fbxEnable := scParameter.scAlCondition.fbxEnable;
END_GET
END_PROPERTY

PROPERTY P_scAlCondition_fbtDelayTillCondition : CtaSysConfig.ITF_DATATYPE
GET
P_scAlCondition_fbtDelayTillCondition := scParameter.scAlCondition.fbtDelayTillCondition;
END_GET
END_PROPERTY

PROPERTY P_scHighAlarm_fbiRetryTillLock : CtaSysConfig.ITF_DATATYPE
GET
P_scHighAlarm_fbiRetryTillLock := scParameter.scHighAlarm.fbiRetryTillLock;
END_GET
END_PROPERTY

PROPERTY P_scHighAlarm_fbiTypeOfAcknolage : CtaSysConfig.ITF_DATATYPE
GET
P_scHighAlarm_fbiTypeOfAcknolage := scParameter.scHighAlarm.fbiTypeOfAcknolage;
END_GET
END_PROPERTY

PROPERTY P_scHighAlarm_fbrHysterese : CtaSysConfig.ITF_DATATYPE
GET
P_scHighAlarm_fbrHysterese := scParameter.scHighAlarm.fbrHysterese;
END_GET
END_PROPERTY

PROPERTY P_scHighAlarm_fbrValue : CtaSysConfig.ITF_DATATYPE
GET
P_scHighAlarm_fbrValue := scParameter.scHighAlarm.fbrValue;
END_GET
END_PROPERTY

PROPERTY P_scHighAlarm_fbtDelayTillAlarm : CtaSysConfig.ITF_DATATYPE
GET
P_scHighAlarm_fbtDelayTillAlarm := scParameter.scHighAlarm.fbtDeleayTillAlarm;
END_GET
END_PROPERTY

PROPERTY P_scHighAlram_fbxDoesAlarm : CtaSysConfig.ITF_DATATYPE
GET
P_scHighAlram_fbxDoesAlarm := scParameter.scHighAlarm.fbxDoesAlarm;
END_GET
END_PROPERTY

PROPERTY P_scHighWarning_fbrValue : CtaSysConfig.ITF_DATATYPE
GET
P_scHighWarning_fbrValue := scParameter.scHighWarning.fbrValue;
END_GET
END_PROPERTY

PROPERTY P_scHighWarning_fbtDelayTillWarning : CtaSysConfig.ITF_DATATYPE
GET
P_scHighWarning_fbtDelayTillWarning := scParameter.scHighWarning.fbtDelayTillWarning;
END_GET
END_PROPERTY

PROPERTY P_scHighWarning_fbxDoesWarning : CtaSysConfig.ITF_DATATYPE
GET
P_scHighWarning_fbxDoesWarning := scParameter.scHighWarning.fbxDoesWarning;
END_GET
END_PROPERTY

PROPERTY P_scInfluxDb_fbxEnable : CtaSysConfig.ITF_DATATYPE
GET
P_scInfluxDb_fbxEnable := scParameter.scInfluxDb.fbxEnable;
END_GET
END_PROPERTY

PROPERTY P_scLoAlarm_fbiRetryTillLock : CtaSysConfig.ITF_DATATYPE
GET
P_scLoAlarm_fbiRetryTillLock := scParameter.scLoAlarm.fbiRetryTillLock;
END_GET
END_PROPERTY

PROPERTY P_scLoAlarm_fbiTypeOfAcknolage : CtaSysConfig.ITF_DATATYPE
GET
P_scLoAlarm_fbiTypeOfAcknolage := scParameter.scLoAlarm.fbiTypeOfAcknolage;
END_GET
END_PROPERTY

PROPERTY P_scLoAlarm_fbrHysterese : CtaSysConfig.ITF_DATATYPE
GET
P_scLoAlarm_fbrHysterese := scParameter.scLoAlarm.fbrHysterese;
END_GET
END_PROPERTY

PROPERTY P_scLoAlarm_fbrValue : CtaSysConfig.ITF_DATATYPE
GET
P_scLoAlarm_fbrValue := scParameter.scLoAlarm.fbrValue;
END_GET
END_PROPERTY

PROPERTY P_scLoAlarm_fbtDelayTillAlarm : CtaSysConfig.ITF_DATATYPE
GET
P_scLoAlarm_fbtDelayTillAlarm := scParameter.scLoAlarm.fbtDeleayTillAlarm;
END_GET
END_PROPERTY

PROPERTY P_scLoAlarm_fbxDoesAlarm : CtaSysConfig.ITF_DATATYPE
GET
P_scLoAlarm_fbxDoesAlarm := scParameter.scLoAlarm.fbxDoesAlarm;
END_GET
END_PROPERTY

PROPERTY P_scLoWarning_fbrValue : CtaSysConfig.ITF_DATATYPE
GET
P_scLoWarning_fbrValue := scParameter.scLoWarning.fbrValue;
END_GET
END_PROPERTY

PROPERTY P_scLoWarning_fbtDelayTillWarning : CtaSysConfig.ITF_DATATYPE
GET
P_scLoWarning_fbtDelayTillWarning := scParameter.scLoWarning.fbtDelayTillWarning;
END_GET
END_PROPERTY

PROPERTY P_scLoWarning_fbxDoesWarning : CtaSysConfig.ITF_DATATYPE
GET
P_scLoWarning_fbxDoesWarning := scParameter.scLoWarning.fbxDoesWarning;
END_GET
END_PROPERTY

PROPERTY P_scManual_fbrManualOnY : CtaSysConfig.ITF_DATATYPE
GET
P_scManual_fbrManualOnY := scParameter.scManual.fbrManualOnY;
END_GET
END_PROPERTY

PROPERTY P_scManual_fbuiManualControl : CtaSysConfig.ITF_DATATYPE
GET
P_scManual_fbuiManualControl := scParameter.scManual.fbuiManualControl;
END_GET
END_PROPERTY

PROPERTY P_scManual_fbuiManualState : CtaSysConfig.ITF_DATATYPE
GET
P_scManual_fbuiManualState := scParameter.scManual.fbuiManualState;
END_GET
END_PROPERTY

PROPERTY P_scManual_fbxAllowManualOn : CtaSysConfig.ITF_DATATYPE
GET
P_scManual_fbxAllowManualOn := scParameter.scManual.fbxAlowManualOn;
END_GET
END_PROPERTY

PROPERTY P_scAlarmReset_fbtDealyTillReset : CtaSysConfig.ITF_DATATYPE
GET
P_scAlarmReset_fbtDealyTillReset := scParameter.scAlarmReset.fbtDelayTillReset;
END_GET
END_PROPERTY

PROPERTY P_scFilter_fbrValue : CtaSysConfig.ITF_DATATYPE
GET
P_scFilter_fbrValue := scParameter.scFilter.fbrValue;
END_GET
END_PROPERTY

PROPERTY P_scFilter_fbxEnabled : CtaSysConfig.ITF_DATATYPE
GET
P_scFilter_fbxEnabled := scParameter.scFilter.fbxEnabled;
END_GET
END_PROPERTY

PROPERTY proSensorITF : CtaSysIO.ITF_IO;
GET
proSensorITF := ITF_IO_IN;
END_GET
END_PROPERTY

PROPERTY proRawValue : STRING
GET
IF xIsITF THEN
	IF __QUERYINTERFACE (_ITF_DI,_ITF_DI) THEN	
		proRawValue := TO_STRING(_ITF_DI.proValue);
	ELSIF __QUERYINTERFACE(_ITF_AI,_ITF_AI) THEN
		IF _ITF_AI.IO_TYPE = CtaSysIO.enIOType.DC_0_10V_IN THEN
			proRawValue :=	CONCAT(TO_STRING(_ITF_AI.proPhysicalValue),' v');
		ELSIF _ITF_AI.IO_TYPE = CtaSysIO.enIOType.DC_4_20mA_IN THEN
			proRawValue :=	CONCAT(TO_STRING(_ITF_AI.proPhysicalValue),' mA');
		ELSIF _ITF_AI.IO_TYPE = CtaSysIO.enIOType.TEMPERATUR THEN
			proRawValue :=	CONCAT(TO_STRING(_ITF_AI.proPhysicalValue),' °C');
		ELSE
			proRawValue := '';	
		END_IF
	ELSE
		proRawValue := '';			
	END_IF	
ELSIF xIsBool THEN
	proRawValue := TO_STRING(xValueIn);
ELSIF xIsReal THEN
	proRawValue := TO_STRING(rValueIn);
ELSE
	proRawValue := '';	
END_IF
END_GET
END_PROPERTY

PROPERTY proSoftwareValue : STRING
GET
IF xIsBool OR ( xIsITF AND __QUERYINTERFACE (_ITF_DI,_ITF_DI)) THEN
	proSoftwareValue := TO_STRING(xValue);
ELSIF xIsReal THEN
	proSoftwareValue := CONCAT(TO_STRING(CTASYsCONFIG.fcRealToString(rValue,scparameter.scVisu.fbusiDezimalPos.usiValue)),stAlternateUnit);	 
ELSIF xIsITF AND __QUERYINTERFACE(_ITF_AI,_ITF_AI) THEN
	IF _ITF_AI.IO_TYPE = CtaSysIO.enIOType.TEMPERATUR THEN
		proSoftwareValue := CONCAT(TO_STRING(CTASYsCONFIG.fcRealToString(rValue,scparameter.scVisu.fbusiDezimalPos.usiValue)),'°C') ;
	ELSE
		proSoftwareValue := CONCAT(TO_STRING(CTASYsCONFIG.fcRealToString(rValue,scparameter.scVisu.fbusiDezimalPos.usiValue)),CtaSysConfig.fcGetValueFromDataType(_ITF_AI.P_scfbAI_fbstPhysicalUnit)) ;
	END_IF	
ELSE
	proSoftwareValue := '';
END_IF
END_GET
END_PROPERTY

PROPERTY proIsWarning : BOOL
GET
proIsWarning := xIsWarning;
END_GET
END_PROPERTY

PROPERTY proIsHandOnOrOff : BOOL
GET
proIsHandOnOrOff := xIsHand;
END_GET
END_PROPERTY

PROPERTY proIsReady : BOOL
GET
proIsReady := xIsEnabled AND NOT xIsError;
END_GET
END_PROPERTY

PROPERTY proHandOff : BOOL
SET
IF proHandOff THEN
	scParameter.scManual.fbuiManualState.proValue := 1;
END_IF
END_SET
GET
proHandOff := xIsHandOff;
END_GET
END_PROPERTY

PROPERTY proHandOn : BOOL
GET
proHandOn := xIsHandOn OR xIsHandMode;
END_GET
SET
IF proHandOn THEN
	scParameter.scManual.fbuiManualState.proValue := 2;
END_IF
END_SET
END_PROPERTY

PROPERTY proHandOnY : REAL
SET
scParameter.scManual.fbrManualOnY.proValue := proHandOnY;
END_SET
GET
proHandOnY := scParameter.scManual.fbrManualOnY.proValue;
END_GET
END_PROPERTY

PROPERTY proAuto : BOOL
SET
IF proAuto THEN
	scParameter.scManual.fbuiManualState.provalue := 0;
END_IF
END_SET
GET
proAuto := xIsAuto;
END_GET
END_PROPERTY

PROPERTY proManualTrue : BOOL
SET
IF proManualTrue THEN
	scParameter.scManual.fbuiManualControl.proValue := 1;
END_IF
END_SET
GET
proManualTrue := xManualValue;
END_GET
END_PROPERTY

PROPERTY proManualFalse : BOOL
SET
IF proManualFalse THEN
	scParameter.scManual.fbuiManualControl.proValue := 0;
END_IF
END_SET
GET
proManualFalse := NOT xManualValue;
END_GET
END_PROPERTY

PROPERTY proValueInputType : enInputType
GET
proValueInputType := enValueInputType;
END_GET
END_PROPERTY

METHOD metSetITF
VAR_INPUT
	ITF_IN		:	CtaSysIO.ITF_IO;
END_VAR
ITF_IO_IN := ITF_IN;
xIsITF 	:= TRUE;
xIsBool := FALSE;
xIsReal := FALSE;
END_METHOD

ACTION actDigital:
IF _ITF_DI <> 0 THEN
	xValueTemp := _ITF_DI.proValue;
ELSE
	xValueTemp := xValueIn;	
END_IF

(* Low Controll *)
xLoWarning      := fcLowControl(xEn   := scParameter.scLoWarning.fbxDoesWarning.proValue,
								rIst  := TO_REAL(xValueTemp),
								rLow  := 0,
								rHyst := 0,
								xTrig := 0);
								
xLoAlarm      	:= fcLowControl(xEn   := scParameter.scLoAlarm.fbxDoesAlarm.proValue,
								rIst  := TO_REAL(xValueTemp),
								rLow  := 0,
								rHyst := 0,
								xTrig := 0);

(* High Controll *)
xHiWarning     := fcHighControl(xEn   := scParameter.scHighWarning.fbxDoesWarning.proValue,
								rIst  := TO_REAL(xValueTemp),
								rHigh := 1,
								rHyst := 0,
								xTrig := 0);
								
xHiAlarm       := fcHighControl(xEn   := scParameter.scHighAlarm.fbxDoesAlarm.proValue,
								rIst  := TO_REAL(xValueTemp),
								rHigh := 1,
								rHyst := 0,
								xTrig := 0);

(* Hand Off *)
IF scParameter.scManual.fbuiManualState.proValue = 1 THEN
	xValue := NOT xValueTemp;	
	xIsHandMode := FALSE;
(* Hand On *)	
ELSIF scParameter.scManual.fbuiManualState.proValue <> 2 AND NOT xEnHandMode THEN
	(* Value *)
	xValue := xValueTemp;
	xIsHandMode := FALSE;
ELSE
	xValue := SEL(xEnHandMode,xManualValue,TO_BOOL(rSimValue));
	xIsHandMode := TRUE;
	
	IF NOT scParameter.scManual.fbxAlowManualOn.proValue AND NOT xEnHandMode THEN
		xValue := xValueTemp;
		xIsHandMode := FALSE;
	END_IF
END_IF

rValue := TO_REAL(xValue);
END_ACTION

ACTION actAnalog:
IF _ITF_AI <> 0 THEN	
	rValueUngefiltert      := _ITF_AI.proValue;
	xOk					   := _ITF_AI.proOK; 
ELSE	
	rValueUngefiltert      := rValueIn; 
END_IF
        
(* Low Controll *)
xLoWarning	:= fcLowControl(xEn   := scParameter.scLoWarning.fbxDoesWarning.proValue,
							rIst  := rValueUngefiltert,
							rLow  := scParameter.scLoWarning.fbrValue.proValue,
							rHyst := 0,
							xTrig := 0);
(* ToLow Controll *)
xLoAlarm    := fcLowControl(xEn   := scParameter.scLoAlarm.fbxDoesAlarm.proValue,
							rIst  := rValueUngefiltert,
							rlow  := scParameter.scLoAlarm.fbrValue.proValue,
							rHyst := scParameter.scLoAlarm.fbrHysterese.proValue,
							xTrig := xLoAlarm);
							
(* High Controll *)
xHiWarning := fcHighControl(xEn   := scParameter.scHighWarning.fbxDoesWarning.proValue,
							rIst  := rValueUngefiltert,
							rHigh := scParameter.scHighWarning.fbrValue.proValue,
							rHyst := 0,
							xTrig := 0);
(* ToHigh Controll *)
xHiAlarm   := fcHighControl(xEn   := scParameter.scHighAlarm.fbxDoesAlarm.proValue,
							rIst  := rValueUngefiltert,
							rHigh := scParameter.scHighAlarm.fbrValue.proValue,
							rHyst := scParameter.scHighAlarm.fbrHysterese.proValue,
							xTrig := xHiAlarm);
							
(* Filter *)
IF scParameter.scFilter.fbxEnabled.proValue THEN
	fbFilter   				   (rIn  	:= rValueUngefiltert,
								rFilter := scParameter.scFilter.fbrValue.proValue);
	(* Value Out*)
	rValueTemp  := fbFilter.rOut;
ELSE
	(* Value Out*)
	rValueTemp  := rValueUngefiltert;
END_IF

IF scParameter.scManual.fbuiManualState.proValue = 1 THEN
	rValue := 0;
	xIsHandMode := FALSE;
ELSIF scParameter.scManual.fbuiManualState.proValue <> 2 AND NOT xEnHandMode THEN
	rValue := rValueTemp;
	xIsHandMode := FALSE;
ELSE
	rValue := SEL(xEnHandMode,scParameter.scManual.fbrManualOnY.proValue,rSimValue);
	xIsHandMode := TRUE;
	
	IF NOT scParameter.scManual.fbxAlowManualOn.proValue AND NOT xEnHandMode THEN
		rValue := rValueTemp;
		xIsHandMode := FALSE;
	END_IF
END_IF

xValue  := scEWI.iError = 0 AND SEL(_ITF_AI <> 0,TRUE ,xOk);
END_ACTION

PROPERTY proPhysicalValue : STRING
GET
IF xIsITF THEN
	IF __QUERYINTERFACE (_ITF_AI,_ITF_AI)THEN
		proPhysicalValue := CONCAT(TO_STRING(_ITF_AI.proValue),CtaSysConfig.fcGetValueFromDataType(_ITF_AI.P_scfbAI_fbstPhysicalUnit));
	ELSIF __QUERYINTERFACE (_ITF_DI,_ITF_DI) THEN
		proPhysicalValue := TO_STRING(_ITF_DI.proValue);
	ELSE
		proPhysicalValue := '';
	END_IF
ELSIF xIsBool THEN
	proPhysicalValue := TO_STRING(xValueIn);
ELSIF xIsReal THEN
	proPhysicalValue :=TO_STRING(rValueIn);
ELSE
	proPhysicalValue := '';
END_IF
END_GET
END_PROPERTY

ACTION actReCalculate:
IF __QUERYINTERFACE(ITF_RC_QUERY,ITF_RC_QUERY) THEN
	ITF_RC_QUERY.VALUE := rValue;
	rValueRC := ITF_RC_QUERY.CALCULATET_VALUE;
ELSE
	rValueRC := rValue;
END_IF;
END_ACTION

PROPERTY ITF_RC : CtaSysSensorReCalculation.ITF_SENSOR_RE_CALCULATE
SET
ITF_RC_QUERY := ITF_RC;
END_SET
GET
ITF_RC := ITF_RC_QUERY;
END_GET
END_PROPERTY

ACTION actMbState:
IF NOT xModbusTest THEN
    (* State Word 0 Digital Info*)
    ayMbStateWord[0].00     := xValue;
    ayMbStateWord[0].01     := FALSE;
    ayMbStateWord[0].02     := FALSE;
    ayMbStateWord[0].03     := FALSE;
    ayMbStateWord[0].04     := FALSE;
    ayMbStateWord[0].05     := FALSE;
    ayMbStateWord[0].06     := FALSE;
    ayMbStateWord[0].07     := FALSE;
    ayMbStateWord[0].08     := xIsHand;
    ayMbStateWord[0].09     := xIsAuto;
    ayMbStateWord[0].10     := FALSE;
    ayMbStateWord[0].11     := FALSE;
    ayMbStateWord[0].12     := FALSE;
    ayMbStateWord[0].13     := FALSE;
    ayMbStateWord[0].14     := xIsWarning;
    ayMbStateWord[0].15     := xIsError;
	
	IF (enValueInputType = enInputType.DigitalInput) OR (enValueInputType = enInputType.Digital_ITF_Input) THEN
		(* State Word 1 setpoint*)
		ayMbStateWord[1]   	:= TO_WORD(TO_INT(xValue));
		(* State Word 2 actual value*)
		ayMbStateWord[3]	:= TO_WORD(TO_INT(xValue));
	ELSE
		 (* State Word 1 setpoint*)
		ayMbStateWord[1]   	:= TO_WORD(TO_INT(rValue * 10));
		(* State Word 2 actual value*)
		ayMbStateWord[2]	:= TO_WORD(TO_INT(rValueRC * 10));
		(* State Word 3 actual value*)
		ayMbStateWord[3]	:=	SEL(enValueInputType = enInputType.Analog_ITF_Input,TO_WORD(TO_INT(rValue * 10)),TO_WORD(TO_INT(_ITF_AI.proPhysicalValue * 10)));	
	END_IF
END_IF;
END_ACTION

PROPERTY proModbusTest : BOOL
SET
xModbusTest := proModbusTest;
END_SET
GET
proModbusTest := xModbusTest;
END_GET
END_PROPERTY

{warning disable C0410}
PROPERTY proModbusStateWord : REFERENCE TO ARRAY[0..3] OF WORD
{warning restore C0410}
GET
proModbusStateWord REF= ayMbStateWord;
END_GET
END_PROPERTY

{warning disable C0410}
PROPERTY proModbusControllWord : REFERENCE TO ARRAY[0..3] OF WORD
{warning restore C0410}
GET
proModbusControllWord REF= ayMbControllWord;
END_GET
END_PROPERTY

PROPERTY prorValue : REAL
GET
prorValue := rValue;
END_GET
END_PROPERTY

END_FUNCTION_BLOCK

// 21 Interface/ITF_SENSOR
INTERFACE ITF_SENSOR EXTENDS CtaAppBmk.ITF_BMK , CtaAppModbusSpezifikation.ITF_MODBUS_SPEZIFIKATION

{attribute 'hide'} 
PROPERTY proConfigError : BOOL
GET
END_GET
END_PROPERTY

PROPERTY P_scBase_fbxEnable : CtaSysConfig.ITF_DATATYPE
GET
END_GET
END_PROPERTY

PROPERTY P_scVisu_fbusiDezimalPos : CtaSysConfig.ITF_DATATYPE
GET
END_GET
END_PROPERTY

PROPERTY P_scManual_fbxAllowManualOn : CtaSysConfig.ITF_DATATYPE
GET
END_GET
END_PROPERTY

PROPERTY P_scManual_fbuiManualState : CtaSysConfig.ITF_DATATYPE
GET
END_GET
END_PROPERTY

PROPERTY P_scManual_fbuiManualControl : CtaSysConfig.ITF_DATATYPE
GET
END_GET
END_PROPERTY

PROPERTY P_scManual_fbrManualOnY : CtaSysConfig.ITF_DATATYPE
GET
END_GET
END_PROPERTY

PROPERTY P_scFilter_fbxEnabled : CtaSysConfig.ITF_DATATYPE
GET
END_GET
END_PROPERTY

PROPERTY P_scFilter_fbrValue : CtaSysConfig.ITF_DATATYPE
GET
END_GET
END_PROPERTY

PROPERTY P_scLoWarning_fbxDoesWarning : CtaSysConfig.ITF_DATATYPE
GET
END_GET
END_PROPERTY

PROPERTY P_scLoWarning_fbrValue : CtaSysConfig.ITF_DATATYPE
GET
END_GET
END_PROPERTY

PROPERTY P_scLoWarning_fbtDelayTillWarning : CtaSysConfig.ITF_DATATYPE
GET
END_GET
END_PROPERTY

PROPERTY P_scLoAlarm_fbxDoesAlarm : CtaSysConfig.ITF_DATATYPE
GET
END_GET
END_PROPERTY

PROPERTY P_scLoAlarm_fbrValue : CtaSysConfig.ITF_DATATYPE
GET
END_GET
END_PROPERTY

PROPERTY P_scLoAlarm_fbrHysterese : CtaSysConfig.ITF_DATATYPE
GET
END_GET
END_PROPERTY

PROPERTY P_scLoAlarm_fbtDelayTillAlarm : CtaSysConfig.ITF_DATATYPE
GET
END_GET
END_PROPERTY

PROPERTY P_scLoAlarm_fbiRetryTillLock : CtaSysConfig.ITF_DATATYPE
GET
END_GET
END_PROPERTY

PROPERTY P_scLoAlarm_fbiTypeOfAcknolage : CtaSysConfig.ITF_DATATYPE
GET
END_GET
END_PROPERTY

PROPERTY P_scHighWarning_fbxDoesWarning : CtaSysConfig.ITF_DATATYPE
GET
END_GET
END_PROPERTY

PROPERTY P_scHighWarning_fbrValue : CtaSysConfig.ITF_DATATYPE
GET
END_GET
END_PROPERTY

PROPERTY P_scHighWarning_fbtDelayTillWarning : CtaSysConfig.ITF_DATATYPE
GET
END_GET
END_PROPERTY

PROPERTY P_scHighAlram_fbxDoesAlarm : CtaSysConfig.ITF_DATATYPE
GET
END_GET
END_PROPERTY

PROPERTY P_scHighAlarm_fbrValue : CtaSysConfig.ITF_DATATYPE
GET
END_GET
END_PROPERTY

PROPERTY P_scHighAlarm_fbrHysterese : CtaSysConfig.ITF_DATATYPE
GET
END_GET
END_PROPERTY

PROPERTY P_scHighAlarm_fbtDelayTillAlarm : CtaSysConfig.ITF_DATATYPE
GET
END_GET
END_PROPERTY

PROPERTY P_scHighAlarm_fbiRetryTillLock : CtaSysConfig.ITF_DATATYPE
GET
END_GET
END_PROPERTY

PROPERTY P_scHighAlarm_fbiTypeOfAcknolage : CtaSysConfig.ITF_DATATYPE
GET
END_GET
END_PROPERTY

PROPERTY P_scInfluxDb_fbxEnable : CtaSysConfig.ITF_DATATYPE
GET
END_GET
END_PROPERTY

PROPERTY P_scAnalogAlarm_fbxEnableOverflowAl : CtaSysConfig.ITF_DATATYPE
GET
END_GET
END_PROPERTY

PROPERTY P_scAnalogAlarm_fbxEnableUnderflowAl : CtaSysConfig.ITF_DATATYPE
GET
END_GET
END_PROPERTY

PROPERTY P_scAlCondition_fbxEnable : CtaSysConfig.ITF_DATATYPE
GET
END_GET
END_PROPERTY

PROPERTY P_scAlCondition_fbtDelayTillCondition : CtaSysConfig.ITF_DATATYPE
GET
END_GET
END_PROPERTY

PROPERTY P_scAlarmReset_fbtDealyTillReset : CtaSysConfig.ITF_DATATYPE
GET
END_GET
END_PROPERTY

PROPERTY proSensorITF : CtaSysIO.ITF_IO;
GET
END_GET
END_PROPERTY

{attribute 'hide'} 
PROPERTY INTERNAL proCountedError : INT
GET
END_GET
END_PROPERTY

{attribute 'hide'} 
PROPERTY INTERNAL proCountedInfo : INT
GET
END_GET
END_PROPERTY

{attribute 'hide'} 
PROPERTY INTERNAL proITF_REPORTMANAGER : CtaAppReport.ITF_REPORTMANAGER
GET
END_GET
END_PROPERTY

{attribute 'hide'} 
PROPERTY INTERNAL proCountedWarning : INT
GET
END_GET
END_PROPERTY

PROPERTY proRawValue : STRING
GET
END_GET
END_PROPERTY

PROPERTY proSoftwareValue : STRING
GET
END_GET
END_PROPERTY

{attribute 'hide'} 
PROPERTY INTERNAL proEnSymbol : STRING
GET
END_GET
END_PROPERTY

{attribute 'hide'} 
PROPERTY INTERNAL proStateSymbol : STRING
GET
END_GET
END_PROPERTY

PROPERTY proIsHandOnOrOff : BOOL
GET
END_GET
END_PROPERTY

PROPERTY proHandOn : BOOL
SET
END_SET
GET
END_GET
END_PROPERTY

PROPERTY proIsError : BOOL
GET
END_GET
END_PROPERTY

PROPERTY proIsWarning : BOOL
GET
END_GET
END_PROPERTY

PROPERTY proEn : BOOL
GET
END_GET
SET
END_SET
END_PROPERTY

PROPERTY proIsEnabled : BOOL
GET
END_GET
END_PROPERTY

PROPERTY proHandOff : BOOL
SET
END_SET
GET
END_GET
END_PROPERTY

PROPERTY proHandOnY : REAL
SET
END_SET
GET
END_GET
END_PROPERTY

PROPERTY proIsReady : BOOL
GET
END_GET
END_PROPERTY

PROPERTY proAuto : BOOL
SET
END_SET
GET
END_GET
END_PROPERTY

PROPERTY proManualFalse : BOOL
SET
END_SET
GET
END_GET
END_PROPERTY

PROPERTY proManualTrue : BOOL
SET
END_SET
GET
END_GET
END_PROPERTY

PROPERTY proValueInputType : enInputType
GET
END_GET
END_PROPERTY

PROPERTY proPhysicalValue : STRING
GET
END_GET
END_PROPERTY

PROPERTY proxErrorConditionValue : BOOL;
GET
END_GET
END_PROPERTY

PROPERTY proInvertierung : BOOL
GET
END_GET
END_PROPERTY

PROPERTY prorValue : REAL
GET
END_GET
END_PROPERTY

{attribute 'monitoring' := 'variable'}
PROPERTY proLockDown : BOOL
GET
END_GET
END_PROPERTY

{attribute 'monitoring' := 'variable'}
PROPERTY proAvailable : BOOL
GET
END_GET
END_PROPERTY

{attribute 'monitoring' := 'variable'}
PROPERTY proAcknowlege : BOOL
GET
END_GET
END_PROPERTY

PROPERTY proAtIconNr : UINT
GET
END_GET
SET
END_SET
END_PROPERTY

PROPERTY ITF_RC : CtaSysSensorReCalculation.ITF_SENSOR_RE_CALCULATE
SET
END_SET
GET
END_GET
END_PROPERTY

{warning disable C0410}
PROPERTY proModbusStateWord : REFERENCE TO ARRAY[0..3] OF WORD
{warning restore C0410}
GET
END_GET
END_PROPERTY

{attribute 'hide'} 
PROPERTY INTERNAL proModbusTest : BOOL
GET
END_GET
SET
END_SET
END_PROPERTY

{warning disable C0410}
PROPERTY proModbusControllWord : REFERENCE TO ARRAY[0..3] OF WORD
{warning restore C0410}
GET
END_GET
END_PROPERTY

END_INTERFACE

// 30 Program Organization Units/fc's/AlarmControll/fcLowControl
FUNCTION fcLowControl : BOOL
VAR_INPUT
    xEn         :   BOOL;
    rIst        :   REAL;
    rLow        :   REAL;
    rHyst       :   REAL;
    xTrig       :   BOOL;       
END_VAR
VAR_OUTPUT
END_VAR
VAR
END_VAR

IF xTrig AND xEn THEN
   fcLowControl := rIst <= rLow + rHyst;
ELSIF xEn THEN
   fcLowControl := rIst <= rLow;
ELSE 
   fcLowControl := FALSE;
END_IF;

END_FUNCTION

// 30 Program Organization Units/fc's/AlarmControll/fcHighControl
FUNCTION fcHighControl : BOOL
VAR_INPUT
    xEn         :   BOOL;
    rIst        :   REAL;
    rHigh       :   REAL;
    rHyst       :   REAL;
    xTrig       :   BOOL;
END_VAR

IF xTrig AND xEn THEN
   fcHighControl := rIst >= rHigh - rHyst;
ELSIF xEn THEN
   fcHighControl := rIst >= rHigh;
ELSE
   fcHighControl := FALSE;
END_IF;

END_FUNCTION

// 30 Program Organization Units/fc's/fcGetBigerStringValue
FUNCTION fcGetBigerStringValue : INT
VAR_INPUT
    st1     :   STRING(255);
    st2     :   STRING(255);
END_VAR
VAR
    diFor: DINT;
    diMax: DINT;
END_VAR

IF LEN(st1) > LEN(st2) THEN
    diMax := LEN(st2); 
    fcGetBigerStringValue := 1;
ELSIF LEN(st1) < LEN(st2) THEN
    diMax := LEN(st1);
    fcGetBigerStringValue := 2;     
ELSE
    diMax := LEN(st1);    
END_IF;
FOR diFor := 0 TO  diMax DO
    IF st1[diFor] > st2[diFor] THEN
        fcGetBigerStringValue := 1;  
        EXIT; 
    ELSIF st1[diFor] < st2[diFor] THEN
        fcGetBigerStringValue := 2;  
        EXIT;
    END_IF;
END_FOR;

END_FUNCTION

// 30 Program Organization Units/fc's/Visu/fcCheckQuerryAndIconReturn
FUNCTION fcCheckQuerryAndIconReturn : BOOL
VAR_INPUT
	_ITF_IN			: 	ITF_SENSOR;
	_uiIconNr_IN	:	UINT;
END_VAR

IF __QUERYINTERFACE(_ITF_IN,_ITF_IN) THEN
	fcCheckQuerryAndIconReturn := TRUE;	
	_ITF_IN.proAtIconNr := _uiIconNr_IN;
ELSE
	fcCheckQuerryAndIconReturn :=  FALSE;
END_IF

END_FUNCTION

// 40 Visualizations/POPUP/POPUP_SENSOR
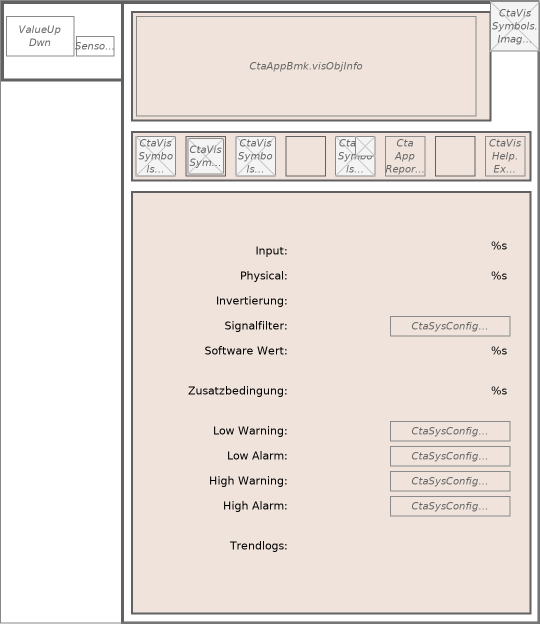
VISUALIZATION POPUP_SENSOR  // 540x624
VAR_INPUT
	ITF_SENSORIN	:	ITF_SENSOR;
	stExklParameter	:	STRING [40];
	uiPopUpGruppe 	: 	UINT;
END_VAR
    RoundedRectangle (1,1 160x80)
    RoundedRectangle (121,1 419x623)
    RoundedRectangle (131,11 360x110)
    RoundedRectangle (131,191 400x423)
    RoundedRectangle (131,131 400x50)
    Frame (136,16 340x100)
        shows CtaAppBmk.visObjInfo(ITF_BMK_IN := ITF_SENSORIN)
    Image (490,1 50x50), image: CtaVisSymbols.ImagePool.close_solo_black
        OnMouseClick:  Dialog=POPUP_SENSOR, Result=None, NumpadKeypadSet=True
    Frame (131,206 399x400), frame switch variable: uiPopUpGruppe
        shows VIS_SENSOR_OVERVIEW(ITF_SENSORIN := ITF_SENSORIN)
        shows VIS_SENSOR_MANUAL(ITF_SENSORIN := ITF_SENSORIN)
        shows VIS_SENSOR_PARAMETER(ITF_SENSORIN := ITF_SENSORIN)
        shows VIS_SENSOR_PLACEHOLDER()
        shows Sensor_BUS(ITF_SENSORIN := ITF_SENSORIN)
        shows VIS_SENSOR_REPORTS(ITF_SENSORIN := ITF_SENSORIN)
        shows VIS_SENSOR_PLACEHOLDER_1()
    Frame (131,136 399x40)
        shows VIS_SENSOR_LISTE(uiPopUpGruppe := uiPopUpGruppe, xHand := ITF_SENSORIN.proIsHandOnOrOff, xHandOff := ITF_SENSORIN.proHandOff, ITF_REPORTMANAGER_IN := ITF_SENSORIN.proITF_REPORTMANAGER, xBusTestAktiv := ITF_SENSORIN.proModbusTest, stExklParameter_IN := stExklParameter)
        pReferences[0]: AnzError=ITF_SENSORIN.proCountedError, AnzWarning=ITF_SENSORIN.proCountedWarning
    Frame (6,16 110x50), input disabled if: TRUE, frame switch variable: ITF_SENSORIN.proAtIconNr
        shows VIS_SENSOR_FLAT_LEFT_ABOVE(ITF_SENSOR_IN := ITF_SENSORIN, stExklParameter := stExklParameter)
        shows VIS_SENSOR_FLAT_LEFT_BELOW(ITF_SENSOR_IN := ITF_SENSORIN, stExklParameter := stExklParameter)
        shows VIS_SENSOR_FLAT_RIGHT_ABOVE(ITF_SENSOR_IN := ITF_SENSORIN, stExklParameter := stExklParameter)
        shows VIS_SENSOR_FLAT_RIGHT_BELOW(ITF_SENSOR_IN := ITF_SENSORIN, stExklParameter := stExklParameter)
        shows VIS_SENSOR_ROUND_RIGHT_ABOVE(ITF_SENSOR_IN := ITF_SENSORIN, stExklParameter := stExklParameter)
        shows VIS_SENSOR_ROUND_RIGHT_BELOW(ITF_SENSOR_IN := ITF_SENSORIN, stExklParameter := stExklParameter)
        shows VIS_SENSOR_ROUND_LEFT_ABOVE(ITF_SENSOR_IN := ITF_SENSORIN, stExklParameter := stExklParameter)
        shows VIS_SENSOR_ROUND_LEFT_BELOW(ITF_SENSOR_IN := ITF_SENSORIN, stExklParameter := stExklParameter)
    InvisibleInput (131,3 360x48)
END_VISUALIZATION

// 40 Visualizations/POPUP/VIS_SENSOR_LISTE
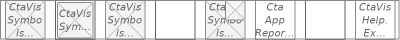
VISUALIZATION VIS_SENSOR_LISTE  // 400x40
VAR_IN_OUT
	uiPopUpGruppe 			:	UINT;
END_VAR
VAR_INPUT
    xHand           		: 	BOOL;
    xHandOff        		: 	BOOL;
    ITF_REPORTMANAGER_IN 	: 	CtaAppReport.ITF_REPORTMANAGER;
    xBusTestAktiv   		: 	BOOL;	
	stExklParameter_IN		:	STRING[40];
END_VAR
    Group (5,0 40x40)
        RoundedRectangle (0,0 40x40), colour toggle: uiPopUpGruppe = 0
            OnMouseDown: execute { uiPopUpGruppe := 0; }
        Image (0,0 40x40), image: CtaVisSymbols.ImagePool.eye
            OnMouseDown: execute { uiPopUpGruppe := 0; }
    Group (55,0 40x40)
        RoundedRectangle (0,0 40x40), colour toggle: uiPopUpGruppe = 1
            OnMouseDown: execute { uiPopUpGruppe := 1; }
        Image (2,2 36x36), image: CtaVisSymbols.ImagePool.front_hand_Black
            OnMouseDown: execute { uiPopUpGruppe := 1; }
        Image (2,2 36x36), invisible if: NOT xHand, image: CtaVisSymbols.ImagePool.front_hand_Yellow
            OnMouseDown: execute { uiPopUpGruppe := 1; }
        Image (2,2 36x36), invisible if: NOT xHandOff, image: CtaVisSymbols.ImagePool.front_hand_Yellow_Off
            OnMouseDown: execute { uiPopUpGruppe := 1; }
    Group (105,0 40x40)
        RoundedRectangle (0,0 40x40), colour toggle: uiPopUpGruppe = 2
            OnMouseDown: execute { uiPopUpGruppe := 2; }
        Image (0,0 40x40), image: CtaVisSymbols.ImagePool.gear
            OnMouseDown: execute { uiPopUpGruppe := 2; }
    Group (155,0 40x40), invisible if: TRUE, input disabled if: TRUE
        RoundedRectangle (0,0 40x40), colour toggle: uiPopUpGruppe = 3, input disabled if: TRUE
            OnMouseDown: execute { uiPopUpGruppe := 3; }
    Group (205,0 40x40)
        RoundedRectangle (0,0 40x40), colour toggle: uiPopUpGruppe = 4
            OnMouseDown: execute { uiPopUpGruppe := 4; }
        Image (0,0 40x40), image: CtaVisSymbols.ImagePool.lan
            OnMouseDown: execute { uiPopUpGruppe := 4; }
        Image (20,0 20x20), invisible if: NOT xBusTestAktiv, image: CtaVisSymbols.ImagePool.front_hand_Yellow
            OnMouseDown: execute { uiPopUpGruppe := 4; }
    Group (255,0 40x40)
        RoundedRectangle (0,0 40x40), colour toggle: uiPopUpGruppe = 5
            OnMouseDown: execute { uiPopUpGruppe := 5; }
        Frame (0,0 40x40), input disabled if: TRUE
            shows CtaAppReport.VIS_ANZ_REPORTS_MODUL(ITF_REPORTMANAGER_IN := ITF_REPORTMANAGER_IN)
            OnMouseDown: execute { uiPopUpGruppe := 5; }
    Group (305,0 40x40), invisible if: TRUE, input disabled if: TRUE
        RoundedRectangle (0,0 40x40), colour toggle: uiPopUpGruppe = 6
            OnMouseDown: execute { uiPopUpGruppe := 6; }
    Group (355,0 40x40)
        RoundedRectangle (0,0 40x40), invisible if: stExklParameter_IN = ' '
        Frame (0,0 40x40)
            shows CtaVisHelp.ExkParameterSymbol(stExklParameter := stExklParameter_IN)
END_VISUALIZATION

// 40 Visualizations/POPUP/PARAMETER/SENSOR_ReportManagement/Sensor_LowAlarm_Param
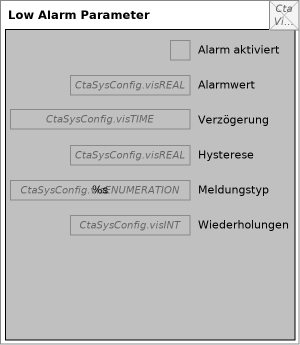
VISUALIZATION Sensor_LowAlarm_Param  // 300x345
VAR_INPUT
	ITF_SENSORIN	:	ITF_SENSOR;
END_VAR
VAR_IN_OUT
    xShow   :   BOOL;
END_VAR
    RoundedRectangle (0,0 299x344)
    RoundedRectangle (5,29 290x311)
    Image (269,0 30x30), image: CtaVisSymbols.ImagePool.close_solo_black
        OnMouseClick: execute { xShow := FALSE; }
    Label (5,0 198x30), "Low Alarm Parameter"
    Label (195,40 100x20), "Alarm aktiviert"
    Frame (170,40 20x20)
        shows CtaSysConfig.visBOOL(visfbBOOLIn := ITF_SENSORIN.P_scLoAlarm_fbxDoesAlarm)
    Label (195,75 100x20), "Alarmwert"
    Frame (70,75 120x20), invisible if: (ITF_SENSORIN.proValueInputType = enInputType.DigitalInput) OR (ITF_SENSORIN.proValueInputType = enInputType.Digital_ITF_Input)
        shows CtaSysConfig.visREAL(visfbREALIn := ITF_SENSORIN.P_scLoAlarm_fbrValue)
    Label (195,110 100x20), "Verzögerung"
    Frame (10,109 180x20)
        shows CtaSysConfig.visTIME(visfbTIMEIn := ITF_SENSORIN.P_scLoAlarm_fbtDelayTillAlarm)
    Frame (70,145 120x20), invisible if: (ITF_SENSORIN.proValueInputType = enInputType.DigitalInput) OR (ITF_SENSORIN.proValueInputType = enInputType.Digital_ITF_Input)
        shows CtaSysConfig.visREAL(visfbREALIn := ITF_SENSORIN.P_scLoAlarm_fbrHysterese)
    Label (195,145 100x20), "Hysterese"
    Frame (10,180 180x20)
        shows CtaSysConfig.visENUMERATION(visfbENUIn := ITF_SENSORIN.P_scLoAlarm_fbiTypeOfAcknolage)
    Label (195,180 100x20), "Meldungstyp"
    Frame (70,215 120x20), invisible if: NOT (CtaSysConfig.fcGetEnumerationId(ITF_SENSORIN.P_scLoAlarm_fbiTypeOfAcknolage) = 2)
        shows CtaSysConfig.visINT(visfbINTIn := ITF_SENSORIN.P_scLoAlarm_fbiRetryTillLock)
    Label (195,215 100x20), "Wiederholungen"
    Textfield (30,180 140x20), "%s", text list: 'CtaAppReport.txtLibAp99_2enTypeOfAck', text index: CtaSysConfig.fcGetEnumerationId(ITF_SENSORIN.P_scLoAlarm_fbiTypeOfAcknolage)
END_VISUALIZATION

// 40 Visualizations/ICON/SENSOR_FLAT/SENSOR_FLAT_TXT_LEFT/ABOVE/VIS_SENSOR_FLAT_LeftAboveCheckQuerry
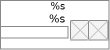
VISUALIZATION VIS_SENSOR_FLAT_LeftAboveCheckQuerry  // 110x50
VAR_INPUT
    ITF_SENSOR_IN   :   ITF_SENSOR;
	stExklParameter	:	STRING [40];	
END_VAR
    Frame (0,0 110x50)
        shows VIS_SENSOR_FLAT_LeftAboveCheckIsEnabled(ITF_SENSOR_IN := ITF_SENSOR_IN, stExklParameter := stExklParameter)
END_VISUALIZATION

// 40 Visualizations/ICON/SENSOR_FLAT/SENSOR_FLAT_TXT_LEFT/ABOVE/VIS_SENSOR_FLAT_LEFT_ABOVE
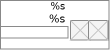
VISUALIZATION VIS_SENSOR_FLAT_LEFT_ABOVE  // 110x50
VAR_INPUT
    ITF_SENSOR_IN   :   ITF_SENSOR;	
END_VAR
VAR_INPUT CONSTANT	
	stExklParameter	:	STRING [40] := ' ';	
END_VAR
VAR CONSTANT
	uiIconNr		: UINT := 0;
END_VAR
    Frame (0,0 110x50), invisible if: NOT fcCheckQuerryAndIconReturn(_ITF_IN := ITF_SENSOR_IN, _uiIconNr_IN := uiIconNr)
        shows VIS_SENSOR_FLAT_LeftAboveCheckQuerry(ITF_SENSOR_IN := ITF_SENSOR_IN, stExklParameter := stExklParameter)
END_VISUALIZATION

// 40 Visualizations/ICON/SENSOR_FLAT/SENSOR_FLAT_TXT_LEFT/ABOVE/VIS_SENSOR_FLAT_LeftAboveCheckIsEnabled
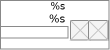
VISUALIZATION VIS_SENSOR_FLAT_LeftAboveCheckIsEnabled  // 110x50
VAR_INPUT
    ITF_SENSOR_IN   :   ITF_SENSOR;
	stExklParameter	:	STRING [40];	
END_VAR
    Frame (70,20 38x20), invisible if: NOT ITF_SENSOR_IN.proIsEnabled
        shows SensorFlat(ITF_SENSORIN := ITF_SENSOR_IN)
    Frame (0,0 68x40), invisible if: NOT ITF_SENSOR_IN.proIsEnabled
        shows ValueUpDwn(ITF_SENSORIN := ITF_SENSOR_IN, uiTextAusrichtung := 6)
    Rectangle (0,0 110x50)
        OnMouseClick:  Dialog=POPUP_SENSOR, Parameters={stExklParameter: stExklParameter, ITF_SENSORIN: ITF_SENSOR_IN, uiPopUpGruppe: 0}, OpenCentered=True
END_VISUALIZATION

// 40 Visualizations/ICON/SENSOR_FLAT/SENSOR_FLAT_TXT_RIGHT/ABOVE/VIS_SENSOR_FLAT_RigthAboveCheckIsEnabled
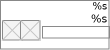
VISUALIZATION VIS_SENSOR_FLAT_RigthAboveCheckIsEnabled  // 110x50
VAR_INPUT
    ITF_SENSOR_IN   :   ITF_SENSOR;
	stExklParameter	:	STRING [40];	
END_VAR
    Frame (2,20 38x20), invisible if: NOT ITF_SENSOR_IN.proIsEnabled
        shows SensorFlat(ITF_SENSORIN := ITF_SENSOR_IN)
    Frame (42,0 68x40), invisible if: NOT ITF_SENSOR_IN.proIsEnabled
        shows ValueUpDwn(ITF_SENSORIN := ITF_SENSOR_IN, uiTextAusrichtung := 4)
    Rectangle (0,0 110x50)
        OnMouseClick:  Dialog=POPUP_SENSOR, Parameters={stExklParameter: stExklParameter, ITF_SENSORIN: ITF_SENSOR_IN, uiPopUpGruppe: 0}, OpenCentered=True
END_VISUALIZATION

// 40 Visualizations/ICON/SENSOR_BASE/ICON/Flat/SensorFlat
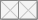
VISUALIZATION SensorFlat  // 38x20
VAR_INPUT
    ITF_SENSORIN   :   ITF_SENSOR;	
END_VAR
    RoundedRectangle (0,0 38x20), colour toggle: ITF_SENSORIN.proAcknowlege, invisible if: ITF_SENSORIN.proIsError
    RoundedRectangle (0,0 38x20), colour toggle: ITF_SENSORIN.proIsError
    Image (0,0 20x20), invisible if: NOT ITF_SENSORIN.proIsWarning, image: CtaVisSymbols.ImagePool.CtaWarning
    Image (18,0 20x20), invisible if: NOT ITF_SENSORIN.proIsHandOnOrOff, image: CtaVisSymbols.ImagePool.front_hand_Yellow
    Image (18,0 20x20), invisible if: NOT ITF_SENSORIN.proHandOff, image: CtaVisSymbols.ImagePool.front_hand_Yellow_Off
END_VISUALIZATION

// 40 Visualizations/POPUP/PARAMETER/VIS_SENSOR_PARAMETER
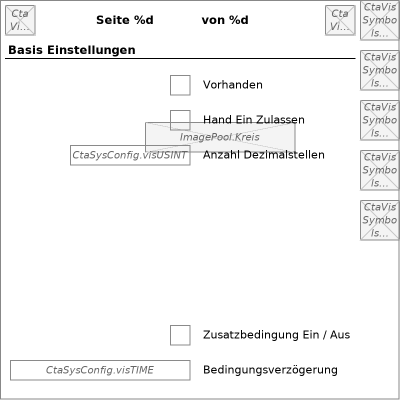
VISUALIZATION VIS_SENSOR_PARAMETER  // 400x400
VAR_INPUT
    ITF_SENSORIN : ITF_SENSOR;
END_VAR
VAR
    uiParameterGruppe : UINT;
END_VAR
    Image (145,122 150x30), image: ImagePool.Kreis
    Frame (360,0 40x300)
        shows VIS_SENSOR_PARAMETER_LISTE(enValueInputType := ITF_SENSORIN.proValueInputType, uiParameterGruppe := uiParameterGruppe)
    Frame (0,0 360x400), frame switch variable: uiParameterGruppe
        shows VIS_SENSOR_PARAMETER_BASE(ITF_SENSORIN := ITF_SENSORIN)
        shows VIS_SENSOR_PARAMETER_FILTER(ITF_SENSORIN := ITF_SENSORIN)
        shows VIS_SENSOR_PARAMETER_REPORTMNG(ITF_SENSORIN := ITF_SENSORIN)
        shows VIS_SENSOR_IO_PARAMETER(ITF_SENSORIN := ITF_SENSORIN)
        shows VIS_SENSOR_PARAMETER_TRENDLOG(ITF_SENSORIN := ITF_SENSORIN)
END_VISUALIZATION

// 40 Visualizations/POPUP/PARAMETER/VIS_SENSOR_PARAMETER_LISTE
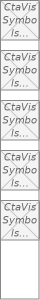
VISUALIZATION VIS_SENSOR_PARAMETER_LISTE  // 40x300
VAR_INPUT
	enValueInputType : enInputType;
END_VAR
VAR_IN_OUT
	uiParameterGruppe : UINT;
END_VAR
    RoundedRectangle (0,150 39x39), colour toggle: uiParameterGruppe = 3, invisible if: enValueInputType = 0 OR enValueInputType = 1 OR enValueInputType = 2, input disabled if: enValueInputType = 0 OR enValueInputType = 1 OR enValueInputType = 2
        OnMouseDown: execute { uiParameterGruppe := 3; }
    RoundedRectangle (0,100 39x39), colour toggle: uiParameterGruppe = 2
        OnMouseDown: execute { uiParameterGruppe := 2; }
    RoundedRectangle (0,50 39x39), colour toggle: uiParameterGruppe = 1
        OnMouseDown: execute { uiParameterGruppe := 1; }
    RoundedRectangle (0,0 39x39), colour toggle: uiParameterGruppe = 0
        OnMouseDown: execute { uiParameterGruppe := 0; }
    RoundedRectangle (0,200 39x39), colour toggle: uiParameterGruppe = 4
        OnMouseDown: execute { uiParameterGruppe := 4; }
    Image (0,0 40x40), image: CtaVisSymbols.ImagePool.Sensor_Black
        OnMouseDown: execute { uiParameterGruppe := 0; }
    Image (0,50 40x40), image: CtaVisSymbols.ImagePool.SearchFilter
        OnMouseDown: execute { uiParameterGruppe := 1; }
    Image (0,100 40x40), image: CtaVisSymbols.ImagePool.notification_black
        OnMouseDown: execute { uiParameterGruppe := 2; }
    Image (0,150 40x40), invisible if: enValueInputType = 0 OR enValueInputType = 1 OR enValueInputType = 2, input disabled if: enValueInputType = 0 OR enValueInputType = 1 OR enValueInputType = 2, image: CtaVisSymbols.ImagePool.dip-switch
        OnMouseDown: execute { uiParameterGruppe := 3; }
    Image (0,200 40x40), image: CtaVisSymbols.ImagePool.sine-wave
        OnMouseDown: execute { uiParameterGruppe := 4; }
END_VISUALIZATION

